// Transition to DURING_MOTION drive mode
rtEnableMode(CLK:=(stMotionStage.nEnableMode = E_StageEnableMode.DURING_MOTION));
// Handle auto-enable timing
CASE stMotionStage.nEnableMode OF
    E_StageEnableMode.ALWAYS:
        stMotionStage.bEnable := TRUE;
    E_StageEnableMode.DURING_MOTION:
        IF rtEnableMode.Q THEN
            stMotionStage.bEnable := FALSE;
        END_IF
        IF bNewMoveReq THEN
            IF stMotionStage.nCommand = E_EpicsMotorCmd.HOME THEN
                stMotionStage.bEnable := stMotionStage.bSafetyReady;
            ELSIF bPosGoal THEN
                IF stMotionStage.bAllForwardEnable THEN
                    stMotionStage.bEnable S= stMotionStage.bSafetyReady;
                ELSIF NOT stMotionStage.bError THEN
                    // Not an error, just a warning
                    stMotionStage.sErrorMessage := 'Cannot move past positive limit.';
                    stMotionStage.bExecute := FALSE;
                END_IF
            ELSIF bNegGoal THEN
                IF stMotionStage.bAllBackwardEnable THEN
                    stMotionStage.bEnable S= stMotionStage.bSafetyReady;
                ELSIF NOT stMotionStage.bError THEN
                    // Not an error, just a warning
                    stMotionStage.sErrorMessage := 'Cannot move past negative limit.';
                    stMotionStage.bExecute := FALSE;
                END_IF
            ELSE
                // Super rare condition where we asked for a move to exactly the same floating point we're already at
                stMotionStage.bEnable S= stMotionStage.bSafetyReady;
            END_IF
            IF stMotionStage.bEnable OR stMotionStage.bError THEN
                bNewMoveReq := FALSE;
            END_IF
        END_IF
END_CASE

// Update all enable booleans
fbSetEnables(stMotionStage:=stMotionStage);

IF stMotionStage.stAxisStatus.bBusy AND NOT bExecute THEN
    // Wait for the previous move to end
    bExecute := FALSE;
ELSIF bMoveCmd THEN
    // Do not start the move until we have power and the safety system says it is OK
    bExecute := stMotionStage.bExecute AND stMotionStage.bAllEnable AND stMotionStage.bEnableDone AND stMotionStage.bSafetyReady;
ELSE
    bExecute := stMotionStage.bExecute;
END_IF

IF bExecute AND NOT stMotionStage.bError THEN
    // Reset local warnings if things are going well
    stMotionStage.sErrorMessage := '';
END_IF

// No moves allowed in error states
IF stMotionStage.bError THEN
    bExecute := FALSE;
END_IF


bExecHome := bExecute AND stMotionStage.nCommand = 10;
bExecMove := bExecute AND NOT bExecHome;

// handles backlash compensention
fbBacklashCompensation(stMotionStage:=stMotionStage,
    bHoming:=bExecHome,
    bMoving:=bExecMove );

// Handle standard commands using ESS's FB
fbDriveVirtual(En:=TRUE,
    bEnable:=stMotionStage.bAllEnable,
    bReset:=stMotionStage.bReset,
    bExecute:=bExecMove,
    nCommand:=INT_TO_UINT(stMotionStage.nCommand),
    nCmdData:=INT_TO_UINT(stMotionStage.nCmdData),
    fVelocity:=stMotionStage.fVelocity,
    fPosition:=stMotionStage.fPosition,
    fAcceleration:=stMotionStage.fAcceleration,
    fDeceleration:=stMotionStage.fDeceleration,
    bLimitFwd:=stMotionStage.bAllForwardEnable,
    bLimitBwd:=stMotionStage.bAllBackwardEnable,
    bHomeSensor:=stMotionStage.bHome,
    fHomePosition:=stMotionStage.fHomePosition,
    bPowerSelf:=stMotionStage.bPowerSelf,
    nMotionAxisID=>stMotionStage.nMotionAxisID,
    Axis:=stMotionStage.Axis);

// Some custom home handling
fbMotionHome(
    stMotionStage:=stMotionStage,
    bExecute:=bExecHome);

// Update status again after the move starts or stops
stMotionStage.Axis.ReadStatus();

// Check for a new error
IF NOT stMotionStage.bError THEN
    stMotionStage.bError := fbDriveVirtual.bError;
    stMotionStage.nErrorId := fbDriveVirtual.nErrorId;
END_IF
IF NOT stMotionStage.bError THEN
    stMotionStage.bError := fbBacklashCompensation.bError;
    stMotionStage.nErrorId := fbBacklashCompensation.nErrorId;
END_IF
IF NOT stMotionStage.bError THEN
    stMotionStage.bError := fbMotionHome.bError;
    stMotionStage.nErrorId := fbMotionHome.nErrorId;
END_IF
IF NOT stMotionStage.bError AND stMotionStage.bExecute AND NOT stMotionStage.bUserEnable THEN
    stMotionStage.bError := TRUE;
    stMotionStage.nErrorId := 1;
    stMotionStage.sCustomErrorMessage := 'Move requested, but user enable is disabled!';
END_IF

// Set the error message if we have one
IF stMotionStage.bError THEN
    // Hook if other code wants to inject a non-NC error
    IF stMotionStage.sCustomErrorMessage <> '' THEN
        stMotionStage.sErrorMessage := stMotionSTage.sCustomErrorMessage;
    ELSE
        stMotionStage.sErrorMessage := F_MotionErrorCodeLookup(nErrorId := stMotionStage.nErrorId);
    END_IF
END_IF

fbLogError(
    stMotionStage:=stMotionStage,
    bEnable:=TRUE);

// When we start, set the busy/done appropriately
rtExec(CLK:=bExecute);
IF rtExec.Q THEN
    stMotionStage.bBusy := TRUE;
    stMotionStage.bDone := FALSE;
END_IF

// Force everything off in case of error
IF stMotionStage.bError THEN
    stMotionStage.bBusy := FALSE;
    stMotionStage.bDone := FALSE;
    stMotionStage.bEnable := FALSE;
END_IF

// Check the limits and cancel execution if appropriate. Without this block we have infinite error spam
bFwdHit := stMotionStage.Axis.Status.PositiveDirection AND NOT stMotionStage.bAllForwardEnable;
bBwdHit := stMotionStage.Axis.Status.NegativeDirection AND NOT stMotionStage.bAllBackwardEnable;
IF (bFwdHit OR bBwdHit) AND NOT fbMotionHome.bBusy THEN
    stMotionStage.bExecute := FALSE;
END_IF

// Check done moving via user stop, fbDriveVirtual and Target Position Monitoring, or from homing.
ftExec(CLK:=stMotionStage.bExecute);
rtTarget(CLK:=(stMotionStage.Axis.Status.InTargetPosition AND fbDriveVirtual.bDone AND bExecMove));
rtHomed(CLK:=fbMotionHome.bDone AND bExecHome);
IF ftExec.Q OR rtTarget.Q OR rtHomed.Q THEN
    IF NOT stMotionStage.bDone THEN
        stMotionStage.bDone := TRUE;
        stMotionStage.bBusy := FALSE;
        IF NOT stMotionStage.Axis.Status.Error THEN
            bExecute := FALSE;
            stMotionStage.bExecute := FALSE;
        END_IF
    END_IF
END_IF

// Handle auto-disable timing
bPrepareDisable S= stMotionStage.nEnableMode = E_StageEnableMode.DURING_MOTION AND ftExec.Q;
// Delay the disable until we reach standstill, else brake issues or other race conditions
IF bPrepareDisable AND stMotionStage.Axis.Status.MotionState = MC_AXISSTATE_STANDSTILL THEN
    bPrepareDisable := FALSE;
    stMotionStage.bEnable := FALSE;
END_IF

// Get a definitive bEnabled reading
CASE stMotionStage.Axis.Status.MotionState OF
    // We are not enabled if there is an issue
    MC_AXISSTATE_UNDEFINED, MC_AXISSTATE_DISABLED, MC_AXISSTATE_ERRORSTOP:
        stMotionStage.bEnableDone := FALSE;
    ELSE
        stMotionStage.bEnableDone := TRUE;
END_CASE

// Handle the brake. TRUE means brake disabled/released
IF stMotionStage.nBrakeMode <> E_StageBrakeMode.NO_BRAKE THEN
    CASE stMotionStage.Axis.Status.MotionState OF
        MC_AXISSTATE_UNDEFINED,
        MC_AXISSTATE_DISABLED,
        MC_AXISSTATE_ERRORSTOP:
            stMotionStage.bBrakeRelease := FALSE;
        MC_AXISSTATE_STANDSTILL:
            IF stMotionStage.nBrakeMode = E_StageBrakeMode.IF_MOVING THEN
                stMotionStage.bBrakeRelease := FALSE;
            ELSE
                stMotionStage.bBrakeRelease := TRUE;
            END_IF
        ELSE
            stMotionStage.bBrakeRelease := TRUE;
    END_CASE
END_IF

// Sync the epics status struct
stMotionStage.stAxisStatus := fbDriveVirtual.stAxisStatus;
stMotionStage.stAxisStatus.bEnabled := stMotionStage.bEnableDone;

// Override homing status, dmov as appropriate
stMotionStage.bHomed := fbMotionHome.bDone AND NOT fbMotionHome.bError;
stMotionStage.stAxisStatus.bHomed := stMotionStage.bHomed;
stMotionStage.stAxisStatus.bExecute := bExecute;
stMotionStage.stAxisStatus.nCommand := 3; // If this is not 3, the IOC stops updating positions during homing

// Fill in auxiliary status info
stMotionStage.fPosDiff := stMotionStage.Axis.NcToPlc.PosDiff;

// Reset everything when bReset is flagged
IF stMotionStage.bReset THEN
    stMotionStage.bEnable := FALSE;
    stMotionStage.bReset := FALSE;
    stMotionStage.bExecute := FALSE;
    stMotionStage.bError := FALSE;
    stMotionStage.nErrorId := 0;
    stMotionStage.sErrorMessage := '';
    stMotionStage.sCustomErrorMessage := '';
    bExecute := FALSE;
END_IF

fbEncoderValue(stMotionStage:=stMotionStage);
fbNCParams(
    stMotionStage:=stMotionStage,
    bEnable:=TRUE,
    tRefreshDelay:=T#1s);

// Save and restore as long as not an absolute encoder
fbSaveRestore(
    stMotionStage:=stMotionStage,
    bEnable:=stMotionStage.nHomingMode <> E_EpicsHomeCmd.NONE);

// Main Motion Status Structure
stMotionStatus.nMotionAxisID    := stMotionStage.Axis.NcToPlc.AxisId;
stMotionStatus.bEnabled         := stMotionStage.bAllEnable;
stMotionStatus.bHomeSensor      := stMotionStage.bHome;
stMotionStatus.bLimitBwd        := stMotionStage.bAllBackwardEnable;
stMotionStatus.bLimitFwd        := stMotionStage.bAllForwardEnable;
stMotionStatus.fActDiff         := stMotionStage.Axis.NcToPlc.PosDiff;
stMotionStatus.fActPosition     := stMotionStage.Axis.NcToPlc.ActPos;
stMotionStatus.fActVelocity     := stMotionStage.Axis.NcToPlc.ActVelo;
stMotionStatus.fOverride        := stMotionStage.Axis.PlcToNc.Override;
stMotionStatus.bBusy            := stMotionStage.bBusy;
stMotionStatus.bHomed           := stMotionStage.bHomed;
stMotionStatus.bWarning         := FALSE; // NOT SUPPORTED BY THIS IMPLEMENTATION
stMotionStatus.bError           := stMotionStage.bError;
stMotionStatus.nErrorId         := stMotionStage.nErrorId;
stMotionStatus.sErrorMessage    := stMotionStage.sErrorMessage;

// Extended Motion Status (Debug, Testing) NOT SUPPORTED BY THIS IMPLEMENTATION
// stExMotionStatus.bMotionAxisError
// stExMotionStatus.nMotionAxisErrorId
// stExMotionStatus.bInterlocksError
// stExMotionStatus.nInterlocksError
// stExMotionStatus.eDriveState
// stExMotionStatus.bAbortDone
// stExMotionStatus.bAborted
// stExMotionStatus.bLimHomeDone
// stExMotionStatus.bDriveWatchDogStatus
// stExMotionStatus.bNewMoveReq
// stExMotionStatus.bEnable
// stExMotionStatus.bIdling

// Main Motion Command Structure
stMotionCmdNow.bHalt := FALSE;
stMotionCmdNow.bHomeCmd := FALSE;
stMotionCmdNow.bMoveCmd := FALSE;
stMotionCmdNow.bReset := FALSE;
stMotionCmdNow.fAcceleration := stMotionStage.fAcceleration;
stMotionCmdNow.fDeceleration := stMotionStage.fDeceleration;
stMotionCmdNow.fHomePosition := stMotionStage.fHomePosition;
//stMotionCmdNow.fJerk := stMotionStage.fJerk; NOT SUPPORTED BY THIS IMPLEMENTATION
stMotionCmdNow.fPosition := stMotionStage.fPosition;
stMotionCmdNow.fVelocity := stMotionStage.fVelocity;
stMotionCmdNow.nCmdData := stMotionStage.nCmdData;
stMotionCmdNow.nCommand := stMotionStage.nCommand;

stMotionCmdPrev := stMotionCmdNow;


METHOD AbsoluteMove
VAR_INPUT
    Position	: LREAL;
    Velocity	: LREAL;
    Acceleration	: LREAL;
    Deceleration	: LREAL;
END_VAR

IF NOT __ISVALIDREF(THIS^.stMotionStageMethods) THEN
    RETURN;
END_IF

THIS^.stMotionStageMethods.fPosition := Position;
THIS^.stMotionStageMethods.fVelocity := Velocity;
THIS^.stMotionStageMethods.fAcceleration := Acceleration;
THIS^.stMotionStageMethods.fDeceleration := Deceleration;
THIS^.stMotionStageMethods.bMoveCmd := TRUE;
END_METHOD


METHOD AbsoluteMoveWithBacklashCompensation
VAR_INPUT
    Position	: LREAL;
    Velocity	: LREAL;
    Acceleration	: LREAL;
    Deceleration	: LREAL;
END_VAR

IF NOT __ISVALIDREF(THIS^.stMotionStageMethods) THEN
    RETURN;
END_IF

THIS^.stMotionStageMethods.fPosition := Position;
THIS^.stMotionStageMethods.fVelocity := Velocity;
THIS^.stMotionStageMethods.fAcceleration := Acceleration;
THIS^.stMotionStageMethods.fDeceleration := Deceleration;
THIS^.stMotionStageMethods.bMoveCmd := TRUE;
END_METHOD


PROPERTY BrakeMode : LCLS_OOPMotion.E_StageBrakeMode
GET

CASE THIS^.stMotionStageMethods.nBrakeMode OF
    E_StageBrakeMode.NO_BRAKE:
        BrakeMode := LCLS_OOPMotion.E_StageBrakeMode.NO_BRAKE;
    E_StageBrakeMode.IF_MOVING:
        BrakeMode := LCLS_OOPMotion.E_StageBrakeMode.IF_MOVING;
    E_StageBrakeMode.IF_ENABLED:
        BrakeMode := LCLS_OOPMotion.E_StageBrakeMode.IF_ENABLED;
END_CASE
END_GET
SET

CASE BrakeMode OF
    LCLS_OOPMotion.E_StageBrakeMode.NO_BRAKE:
        THIS^.stMotionStageMethods.nBrakeMode := E_StageBrakeMode.NO_BRAKE;
    LCLS_OOPMotion.E_StageBrakeMode.IF_MOVING:
        THIS^.stMotionStageMethods.nBrakeMode := E_StageBrakeMode.IF_MOVING;
    LCLS_OOPMotion.E_StageBrakeMode.IF_ENABLED:
        THIS^.stMotionStageMethods.nBrakeMode := E_StageBrakeMode.IF_ENABLED;
END_CASE
END_SET
END_PROPERTY


PROPERTY EnableMode : LCLS_OOPMotion.E_StageEnableMode
GET

CASE THIS^.stMotionStageMethods.nEnableMode OF
    E_StageEnableMode.ALWAYS:
        EnableMode := LCLS_OOPMotion.E_StageEnableMode.ALWAYS;
    E_StageEnableMode.DURING_MOTION:
        EnableMode := LCLS_OOPMotion.E_StageEnableMode.DURING_MOTION;
    E_StageEnableMode.NEVER:
        EnableMode := LCLS_OOPMotion.E_StageEnableMode.NEVER;
END_CASE
END_GET
SET

CASE EnableMode OF
    LCLS_OOPMotion.E_StageEnableMode.ALWAYS:
        THIS^.stMotionStageMethods.nEnableMode := E_StageEnableMode.ALWAYS;
    LCLS_OOPMotion.E_StageEnableMode.DURING_MOTION:
        THIS^.stMotionStageMethods.nEnableMode := E_StageEnableMode.DURING_MOTION;
    LCLS_OOPMotion.E_StageEnableMode.NEVER:
        THIS^.stMotionStageMethods.nEnableMode := E_StageEnableMode.NEVER;
END_CASE
END_SET
END_PROPERTY


PROPERTY ExMotionStatus : REFERENCE TO LCLS_OOPMotion.ST_ExtendedMotionStatus
GET

ExMotionStatus REF= THIS^.stExMotionStatus;
END_GET
END_PROPERTY


METHOD Halt

IF NOT __ISVALIDREF(THIS^.stMotionStageMethods) THEN
    RETURN;
END_IF

THIS^.stMotionStageMethods.bExecute := FALSE;
END_METHOD


METHOD Home
VAR_INPUT
    HomePosition	: LREAL;
    HomeMode	: INT;
END_VAR

IF NOT __ISVALIDREF(THIS^.stMotionStageMethods) THEN
    RETURN;
END_IF

THIS^.stMotionStageMethods.fHomePosition := HomePosition;

CASE HomeMode OF
    E_EpicsHomeCmd.ABSOLUTE_SET:
        THIS^.stMotionStageMethods.nHomingMode := E_EpicsHomeCmd.ABSOLUTE_SET;
    E_EpicsHomeCmd.AutoMethod:
        THIS^.stMotionStageMethods.nHomingMode := E_EpicsHomeCmd.AutoMethod;
    E_EpicsHomeCmd.CURRENT_POSITION_METHOD:
        THIS^.stMotionStageMethods.nHomingMode := E_EpicsHomeCmd.CURRENT_POSITION_METHOD;
    E_EpicsHomeCmd.HIGH_LIMIT:
        THIS^.stMotionStageMethods.nHomingMode := E_EpicsHomeCmd.HIGH_LIMIT;
    E_EpicsHomeCmd.HOME_VIA_HIGH:
        THIS^.stMotionStageMethods.nHomingMode := E_EpicsHomeCmd.HOME_VIA_HIGH;
    E_EpicsHomeCmd.HOME_VIA_LOW:
        THIS^.stMotionStageMethods.nHomingMode := E_EpicsHomeCmd.HOME_VIA_LOW;
    E_EpicsHomeCmd.LOW_LIMIT:
        THIS^.stMotionStageMethods.nHomingMode := E_EpicsHomeCmd.LOW_LIMIT;
    E_EpicsHomeCmd.NONE:
        THIS^.stMotionStageMethods.nHomingMode := E_EpicsHomeCmd.NONE;
END_CASE

THIS^.stMotionStageMethods.bHomeCmd := TRUE;
END_METHOD


PROPERTY MotionCmd : REFERENCE TO LCLS_OOPMotion.ST_MotionCommand
GET

MotionCmd REF= THIS^.stMotionCmdNow;
END_GET
END_PROPERTY


PROPERTY MotionStatus : REFERENCE TO LCLS_OOPMotion.ST_MotionStatus
GET

MotionStatus REF= THIS^.stMotionStatus;
END_GET
END_PROPERTY


METHOD Reset

IF NOT __ISVALIDREF(THIS^.stMotionStageMethods) THEN
    RETURN;
END_IF

THIS^.stMotionStageMethods.bReset := TRUE;
END_METHOD


PROPERTY SaveAxisParams : BOOL
SET

// NOT SUPPORTED BY THIS IMPLEMENTATION
END_SET
END_PROPERTY


METHOD StateMove
VAR_INPUT
    Execute	: BOOL;
END_VAR

IF NOT __ISVALIDREF(stMotionStageMethods) THEN
    RETURN;
END_IF
END_METHOD

END_FUNCTION_BLOCK

// ---- POUs/Motion/FB_MotionHoming.TcPOU
FUNCTION_BLOCK FB_MotionHoming
VAR_IN_OUT
    stMotionStage: ST_MotionStage;
END_VAR
VAR_INPUT
    bExecute: BOOL;
END_VAR
VAR_OUTPUT
    bBusy: BOOL;
    bDone: BOOL;
    bError: BOOL;
    nErrorID: UDINT;
END_VAR
VAR
    fbSetPos: MC_SetPosition;
    fbJog: MC_Jog;
    rtExec: R_TRIG;
    ftExec: F_TRIG;
    nHomeStateMachine: INT := IDLE;
    nStateAfterStop: INT;
    nMoves: INT;
    bFirstDirection: BOOL;
    bAtHome: BOOL;
    bMove: BOOL;
    nErrCount: INT;
    bInterrupted: BOOL;
END_VAR
VAR CONSTANT
    IDLE: INT := 0;
    NEXT_MOVE: INT := 1;
    CHECK_FWD: INT := 2;
    CHECK_BWD: INT := 3;
    FINAL_MOVE: INT := 4;
    FINAL_SETPOS: INT := 5;
    ERROR: INT := 6;
    WAIT_STOP: INT := 7;

    (*
        This is a simpler way of disabling the soft limits that ends up being really obvious if something has gone wrong.
        If you turn the limits off/on, not only do you need to keep track of if you had soft limits set,
        but you need to always restore this properly or risk some issue.
        Instead, I set position to a ridiculous value that can always move forward or backward.
        If this gets stuck for any reason it's very clear that something has gone wrong,
        rather than a silent failure of the soft limit marks.
    *)
    FWD_START: LREAL := -99999999;
    BWD_START: LREAL :=  99999999;
END_VAR


fbSetPos.Options.ClearPositionLag := TRUE;
rtExec(CLK:=bExecute);
ftExec(CLK:=bExecute);

bError R= NOT bExecute;
IF NOT bError THEN
    nErrorID := 0;
END_IF

CASE stMotionStage.nHomingMode OF
    E_EpicsHomeCmd.LOW_LIMIT:
        bFirstDirection := FALSE;
        bAtHome := NOT stMotionStage.bLimitBackwardEnable;
        bMove := TRUE;
    E_EpicsHomeCmd.HIGH_LIMIT:
        bFirstDirection := TRUE;
        bAtHome := NOT stMotionStage.bLimitForwardEnable;
        bMove := TRUE;
    E_EpicsHomeCmd.HOME_VIA_LOW:
        bFirstDirection := FALSE;
        bAtHome := stMotionStage.bHome;
        bMove := TRUE;
    E_EpicsHomeCmd.HOME_VIA_HIGH:
        bFirstDirection := TRUE;
        bAtHome := stMotionStage.bHome;
        bMove := TRUE;
    E_EpicsHomeCmd.ABSOLUTE_SET:
        fbSetPos(
            Axis:=stMotionStage.Axis,
            Execute:=bExecute,
            Position:=stMotionStage.fHomePosition);
        bBusy := rtExec.Q;
        bDone := NOT rtExec.Q;
        bMove := FALSE;
    E_EpicsHomeCmd.NONE:
        bMove := FALSE;
        bBusy := rtExec.Q;
        bDone := NOT rtExec.Q;
    ELSE
        bMove := FALSE;
END_CASE

IF bMove THEN
    IF bBusy AND ftExec.Q THEN
        nHomeStateMachine := ERROR;
        bInterrupted := TRUE;
    END_IF
    CASE nHomeStateMachine OF
        // Wait for a rising edge
        IDLE:
            bBusy := FALSE;
            nErrCount := 0;
            fbSetPos(
                Axis:=stMotionStage.Axis,
                Execute:=FALSE);
            fbJog(
                Axis:=stMotionStage.Axis,
                JogForward:=FALSE,
                JogBackwards:=FALSE);
            IF rtExec.Q THEN
                nHomeStateMachine := NEXT_MOVE;
                nMoves := 0;
                bDone := FALSE;
                bBusy := TRUE;
                bError := FALSE;
                nErrorID := 0;
                bInterrupted := FALSE;
            END_IF
        // Figure out whether to move forward, move backward, or give up
        NEXT_MOVE:
            fbSetPos(
                Axis:=stMotionStage.Axis,
                Execute:=FALSE);
            fbJog(
                Axis:=stMotionStage.Axis,
                JogForward:=FALSE,
                JogBackwards:=FALSE);
            CASE nMoves OF
                0:
                    IF bFirstDirection THEN
                        nStateAfterStop := CHECK_FWD;
                    ELSE
                        nStateAfterStop := CHECK_BWD;
                    END_IF
                1:
                    IF NOT bFirstDirection THEN
                        nStateAfterStop := CHECK_FWD;
                    ELSE
                        nStateAfterStop := CHECK_BWD;
                    END_IF
                ELSE
                    nStateAfterStop := ERROR;
            END_CASE
            nMoves := nMoves + 1;
            IF bAtHome THEN
                nStateAfterStop := FINAL_MOVE;
            END_IF
            nHomeStateMachine := WAIT_STOP;
        // Move forward until we find the home signal or reach end of travel
        CHECK_FWD:
            fbSetPos(
                Axis:=stMotionStage.Axis,
                Execute:=TRUE,
                Position:=FWD_START);
            fbJog(
                Axis:=stMotionStage.Axis,
                JogForward:=stMotionStage.bLimitForwardEnable AND NOT bATHome,
                JogBackwards:=FALSE,
                Mode:=E_JogMode.MC_JOGMODE_CONTINOUS,
                Velocity:=stMotionStage.stAxisParameters.fRefVeloSearch);
            IF NOT fbJog.JogForward THEN
                nHomeStateMachine := NEXT_MOVE;
            ELSIF fbJog.Error THEN
                fbJog(
                    Axis:=stMotionStage.Axis,
                    JogForward:=FALSE,
                    JogBackwards:=FALSE);
                nErrCount := nErrCount + 1;
                IF nErrCount >= 3 THEN
                    nHomeStateMachine := ERROR;
                END_IF
            END_IF
        // Move backward until we find the home signal or reach end of travel
        CHECK_BWD:
            fbSetPos(
                Axis:=stMotionStage.Axis,
                Execute:=TRUE,
                Position:=BWD_START);
            fbJog(
                Axis:=stMotionStage.Axis,
                JogForward:=FALSE,
                JogBackwards:=stMotionStage.bLimitBackwardEnable AND NOT bATHome,
                Mode:=E_JogMode.MC_JOGMODE_CONTINOUS,
                Velocity:=stMotionStage.stAxisParameters.fRefVeloSearch);
            IF NOT fbJog.JogBackwards THEN
                nHomeStateMachine := NEXT_MOVE;
            ELSIF fbJog.Error THEN
                fbJog(
                    Axis:=stMotionStage.Axis,
                    JogForward:=FALSE,
                    JogBackwards:=FALSE);
                nErrCount := nErrCount + 1;
                IF nErrCount >= 3 THEN
                    nHomeStateMachine := ERROR;
                END_IF
            END_IF
        // Set position to get within soft lims, move slowly off signal
        FINAL_MOVE:
            fbSetPos(
                Axis:=stMotionStage.Axis,
                Execute:=TRUE,
                Position:=stMotionStage.fHomePosition);
            IF bAtHome THEN
                fbJog(
                    Axis:=stMotionStage.Axis,
                    JogForward:=NOT bFirstDirection,
                    JogBackwards:=bFirstDirection,
                    Mode:=E_JogMode.MC_JOGMODE_CONTINOUS,
                    Velocity:=stMotionStage.stAxisParameters.fRefVeloSync);
            ELSIF fbJog.Error THEN
                fbJog(
                    Axis:=stMotionStage.Axis,
                    JogForward:=FALSE,
                    JogBackwards:=FALSE);
                nErrCount := nErrCount + 1;
                IF nErrCount >= 3 THEN
                    nHomeStateMachine := ERROR;
                END_IF
            ELSE
                fbJog(
                    Axis:=stMotionStage.Axis,
                    JogForward:=FALSE,
                    JogBackwards:=FALSE);
                fbSetPos(
                    Axis:=stMotionStage.Axis,
                    Execute:=FALSE);
                nHomeStateMachine := WAIT_STOP;
                nStateAfterStop := FINAL_SETPOS;
            END_IF
        FINAL_SETPOS:
            fbSetPos(
                Axis:=stMotionStage.Axis,
                Execute:=TRUE,
                Position:=stMotionStage.fHomePosition);
            nHomeStateMachine := IDLE;
            bBusy := FALSE;
            bDone := TRUE; // need this
        ERROR:
            bError := TRUE;
            nErrorID := fbJog.ErrorID;
            nHomeStateMachine := FINAL_SETPOS;
            fbSetPos(
                Axis:=stMotionStage.Axis,
                Execute:=FALSE);
            IF bInterrupted THEN
                stMotionStage.sCustomErrorMessage := 'Homing interrupted';
            ELSE
                stMotionStage.sCustomErrorMessage := 'Homing failure';
            END_IF
        WAIT_STOP:
            IF stMotionStage.Axis.Status.NotMoving THEN
                nHomeStateMachine := nStateAfterStop;
            END_IF
    END_CASE
END_IF

END_FUNCTION_BLOCK

// ---- POUs/Motion/FB_EncSaveRestore.TcPOU
FUNCTION_BLOCK FB_EncSaveRestore
VAR_IN_OUT
    stMotionStage: ST_MotionStage;
END_VAR
VAR_INPUT
    bEnable: BOOL;
END_VAR
VAR_OUTPUT
END_VAR
VAR
    fbSetPos: MC_SetPosition;
    timer: TON;
    bInit: BOOL;
    bLoad: BOOL;
    nLatchError: UDINT;
    bEncError: BOOL;
    tRetryDelay: TIME := T#1s;
    nMaxRetries: UINT := 10;
    nCurrTries: UINT := 0;
    bWaitRetry: BOOL;
    tonRetry: TON;
END_VAR
VAR PERSISTENT
    bSaved: BOOL;
    fPosition: LREAL;
END_VAR

IF bEnable THEN
    // Trigger a load if anything was saved at all
    IF NOT bInit THEN
        bInit := TRUE;
        bLoad S= bSaved;
        fbSetPos.Options.ClearPositionLag := TRUE;
    END_IF

    // Set our position if bLoad is true
    fbSetPos(
        Axis:=stMotionStage.Axis,
        Execute:=bLoad,
        Position:=fPosition);

    // Only load once, at startup
    bLoad R= fbSetPos.Done OR fbSetPos.Error;

    IF fbSetPos.Error THEN
        // Keep the error latched, it can disappear if Execute is set to FALSE
        nLatchError := fbSetPos.ErrorID;
        nCurrTries := nCurrTries + 1;
        IF nCurrTries >= nMaxRetries THEN
            // Alert the user that something has gone wrong
            stMotionStage.bError := TRUE;
            stMotionStage.nErrorId := nLatchError;
            stMotionStage.sCustomErrorMessage := 'Error loading previously saved position.';
        ELSE
            // Reset the FB for the next retry
            fbSetPos(
                Axis:=stMotionStage.Axis,
                Execute:=FALSE,
                Position:=fPosition);
            // Try again
            bWaitRetry := TRUE;
        END_IF
    END_IF

    tonRetry(
        IN := bWaitRetry,
        PT := tRetryDelay);

    bLoad S= tonRetry.Q;
    bWaitRetry R= tonRetry.Q;

    // Check ST_MotionStage for an encoder error (range 0x44nn)
    bEncError := stMotionStage.bError AND stMotionStage.nErrorId >= 16#4400 AND stMotionStage.nErrorId <= 16#44FF;

    // Do not save if we're currently loading or if there is an encoder error
    IF NOT bLoad AND NOT bEncError AND NOT bWaitRetry THEN
        fPosition := stMotionStage.stAxisStatus.fActPosition;
        // This persistent variable lets us check if anything was saved
        // It will be TRUE at startup if we have saved values
        bSaved := TRUE;
    END_IF
END_IF

END_FUNCTION_BLOCK

// ---- POUs/Motion/FB_LogMotionError.TcPOU
FUNCTION_BLOCK FB_LogMotionError
(*
    If the motion struct has an error, log it.

    The log condition is:
    - When bError goes TRUE (catch transition from no error to error)
    - When the error message changes while bError is TRUE (catch transition from error a to error b)

    Includes the motor name and the NC error id in the json blob
*)
VAR_IN_OUT
    stMotionStage: ST_MotionStage;
END_VAR
VAR_INPUT
    bEnable: BOOL;
END_VAR
VAR
    fbLogMessage: FB_LogMessage;
    rtNewError: R_TRIG;
    bChangedError: BOOL;
    sPrevErr: STRING;
    fbJson: FB_JsonSaxWriter;
END_VAR


rtNewError(CLK:=stMotionStage.bError);
bChangedError := stMotionStage.sErrorMessage <> '' AND stMotionStage.sErrorMessage <> sPrevErr;
sPrevErr := stMotionStage.sErrorMessage;

IF bEnable AND (rtNewError.Q OR bChangedError) THEN
    fbJson.StartObject();
    fbJson.AddKey('schema');
    fbJson.AddString('ST_MotionStage.bError');
    fbJson.AddKey('dut_name');
    fbJson.AddString(stMotionStage.sName);
    fbJson.AddKey('axis_name');
    fbJson.AddString(stMotionStage.stAxisParameters.sAxisName);
    fbJson.AddKey('axis_id');
    fbJson.AddUdint(stMotionStage.stAxisParameters.AxisId);
    fbJson.AddKey('err_id');
    fbJson.AddUdint(stMotionStage.nErrorId);
    fbJson.AddKey('position');
    fbJson.AddLreal(stMotionStage.stAxisStatus.fActPosition);
    fbJson.AddKey('position_lag');
    fbJson.AddLreal(stMotionStage.stAxisStatus.fActDiff);
    fbJson.EndObject();
    fbLogMessage.sJson := fbJson.GetDocument();
    fbLogMessage(
        sMsg := stMotionStage.sErrorMessage,
        eSevr := TcEventSeverity.Error,
        eSubsystem := E_Subsystem.MOTION,
    );
    fbJson.ResetDocument();
END_IF

END_FUNCTION_BLOCK

// ---- POUs/Motion/FB_MotionBacklashCompensation.TcPOU
FUNCTION_BLOCK FB_MotionBacklashCompensation
(*
    Handle positive/negative backlash compensation
    User needs to set the direction of backlash from the sign of the compensation value
    Backlash compensation is disabled during referencing (homing).
    When direction is positive/negative, further movement in the negative/positive direction not compensated
    further movement in the negative/positive direction will be compensated
*)
VAR_IN_OUT
    stMotionStage: ST_MotionStage;
END_VAR
VAR_INPUT
    bHoming: BOOL;
    bMoving: BOOL;
END_VAR
VAR_OUTPUT
    bError: BOOL;
    nErrorID: UDINT;
END_VAR
VAR
    fbBacklashCompensation: MC_BacklashCompensation;
    fPrevCompensation : LREAL := 0.0;
    bBacklashCompEnable: BOOL;
END_VAR

(*Note: Configure within the axis parameters set "position correction" to true *)
(*Directional change for compensation
  default: positive backlash):
  TRUE -> Negative backlash compensation *)
(* Reset Compensation to register a new value change*)
bBacklashCompEnable R= bHoming OR (stMotionStage.fBacklash<>fPrevCompensation);
bBacklashCompEnable S= bMoving;

fbBacklashCompensation(Axis:=stMotionStage.Axis,
    Enable:= ( stMotionStage.bUserBacklashEn AND bBacklashCompEnable),
    Backlash:=stMotionStage.fBacklash,
    CompensationInPositiveDirection:=(stMotionStage.fBacklash<0.0),
    Ramp:=(stMotionStage.fVelocity / 10.0),
    DisableMode:=DisableModeHold,
    Enabled=> stMotionStage.bBacklashStatus,
    Error=>bError,
    ErrorID=>nErrorID,
    CurrentBacklash=>stMotionStage.fCurrentBacklash);

fPrevCompensation:=stMotionStage.fBacklash;

END_FUNCTION_BLOCK

// ---- POUs/Motion/Utils/FB_SetEnables.TcPOU
FUNCTION_BLOCK FB_SetEnables
// Update the all enable booleans based on the booleans that make them up
VAR_IN_OUT
    stMotionStage: ST_MotionStage;
END_VAR

stMotionStage.bAllForwardEnable := stMotionStage.bLimitForwardEnable AND (stMotionStage.bGantryForwardEnable OR NOT stMotionStage.bGantryAxis) AND stMotionStage.stEPSForwardEnable.bEPS_OK;
stMotionStage.bAllBackwardEnable := stMotionStage.bLimitBackwardEnable AND (stMotionStage.bGantryBackwardEnable OR NOT stMotionStage.bGantryAxis) AND stMotionStage.stEPSBackwardEnable.bEPS_OK;

stMotionStage.bAllEnable := stMotionStage.bEnable AND stMotionStage.bHardwareEnable AND stMotionStage.stEPSPowerEnable.bEPS_OK;
stMotionStage.bAllEnable R= NOT stMotionStage.bUserEnable;

END_FUNCTION_BLOCK

// ---- POUs/Motion/FB_EncoderValue.TcPOU
FUNCTION_BLOCK FB_EncoderValue
(*
    Process the encoder value for ST_MotionStage

    A few different problems this is trying to solve:
        1. Different encoders show as different types in the IO,
           but we want a consistent type for checks and for PVs
        2. Some inverted encoders display as very high numbers
           as they count down from max int instead of up from 0
        3. Some encoders have raw signed values, others unsigned.

    To this end, we figure out which encoder is linked and process
    the value appropriately.
*)
VAR_IN_OUT
    stMotionStage: ST_MotionStage;
END_VAR

IF stMotionStage.nRawEncoderULINT <> 0 THEN
    IF stMotionStage.nRawEncoderULINT < 4294967296 THEN
        stMotionStage.nEncoderCount := ULINT_TO_UDINT(stMotionStage.nRawEncoderULINT);
    ELSE
        stMotionStage.nEncoderCount := ULINT_TO_UDINT(18446744073709551615 - stMotionStage.nRawEncoderULINT);
    END_IF
ELSIF stMotionStage.nRawEncoderUINT <> 0 THEN
    stMotionStage.nEncoderCount := UINT_TO_UDINT(stMotionStage.nRawEncoderUINT);
ELSIF stMotionStage.nRawEncoderINT <> 0 THEN
    stMotionStage.nEncoderCount := INT_TO_UDINT(stMotionStage.nRawEncoderINT);
ELSIF stMotionStage.nRawEncoderDINT <> 0 THEN
    stMotionStage.nEncoderCount := DINT_TO_UDINT(stMotionStage.nRawEncoderDINT);
ELSE
    stMotionStage.nEncoderCount := 0;
END_IF

END_FUNCTION_BLOCK

// ---- POUs/Motion/FB_MotionStageNCParams.TcPOU
FUNCTION_BLOCK FB_MotionStageNCParams
(*
    Read and refresh axis parameters struct on ST_MotionStage
*)
VAR_IN_OUT
    stMotionStage: ST_MotionStage;
END_VAR
VAR_INPUT
    bEnable: BOOL;
    tRefreshDelay: TIME;
END_VAR
VAR_OUTPUT
    bError: BOOL;
END_VAR
VAR
    mcReadParams: MC_ReadParameterSet;
    timer: TON;
    bExecute: BOOL := TRUE;
    nLatchErrId: UDINT;
END_VAR

timer(
    IN:=bEnable AND NOT bExecute,
    PT:=tRefreshDelay);
bExecute S= timer.Q;
mcReadParams(
    Parameter:=stMotionStage.stAxisParameters,
    Axis:=stMotionStage.Axis,
    Execute:=bEnable AND bExecute,
    Error=>bError);

// Copy axis parameters that we want to expose to the EPICS layer.
stMotionStage.stAxisParametersExposed.bCtrlEnablePosDiffControl     := stMotionStage.stAxisParameters.bCtrlEnablePosDiffControl;
stMotionStage.stAxisParametersExposed.bEncEnableSoftEndMaxControl   := stMotionStage.stAxisParameters.bEncEnableSoftEndMaxControl;
stMotionStage.stAxisParametersExposed.bEncEnableSoftEndMinControl   := stMotionStage.stAxisParameters.bEncEnableSoftEndMinControl;
stMotionStage.stAxisParametersExposed.fAccelerationMax              := stMotionStage.stAxisParameters.fAccelerationMax;
stMotionStage.stAxisParametersExposed.fCtrlPosDiffMax               := stMotionStage.stAxisParameters.fCtrlPosDiffMax;
stMotionStage.stAxisParametersExposed.fCtrlPosDiffMaxTime           := stMotionStage.stAxisParameters.fCtrlPosDiffMaxTime;
stMotionStage.stAxisParametersExposed.fDecelerationMax              := stMotionStage.stAxisParameters.fDecelerationMax;
stMotionStage.stAxisParametersExposed.fEncSoftEndMax                := stMotionStage.stAxisParameters.fEncSoftEndMax;
stMotionStage.stAxisParametersExposed.fEncSoftEndMin                := stMotionStage.stAxisParameters.fEncSoftEndMin;
stMotionStage.stAxisParametersExposed.fVeloMaximum                  := stMotionStage.stAxisParameters.fVeloMaximum;
stMotionStage.stAxisParametersExposed.fEncOffset               		:= stMotionStage.stAxisParameters.fEncOffset;
stMotionStage.stAxisParametersExposed.fEncScaleFactorInternal       := stMotionStage.stAxisParameters.fEncScaleFactorInternal;

IF mcReadParams.ErrorID <> 0 THEN
    nLatchErrId := 0;
END_IF
bExecute R= mcReadParams.Done OR mcReadParams.Error;
stMotionStage.bAxisParamsInit S= mcReadParams.Done;

END_FUNCTION_BLOCK

// ---- POUs/Motion/Utils/F_MotionErrorCodeLookup.TcPOU
FUNCTION F_MotionErrorCodeLookup : STRING
VAR_INPUT
    nErrorId: UDINT;
END_VAR
VAR
    msg: STRING;
END_VAR

CASE nErrorId OF
    // General NC Errors
    16#4000: msg:='Internal error';
    16#4001: msg:='Memory error';
    16#4002: msg:='Nc retain data error (persistent data)';
    16#4003: msg:='Parameter for Monitoring the NC Setpoint Issuing is Invalid';
    16#4004: msg:='External Error';
    16#4010: msg:='Channel identifier not allowed';
    16#4011: msg:='Group identifier not allowed';
    16#4012: msg:='Axis identifier not allowed';
    16#4013: msg:='Encoder identifier not allowed';
    16#4014: msg:='Controller identifier not allowed';
    16#4015: msg:='Drive identifier not allowed';
    16#4016: msg:='Table identifier not allowed';
    16#4020: msg:='No process image: No PLC-axis interface';
    16#4021: msg:='No process image: No axis-PLC interface';
    16#4022: msg:='No process image: No encoder-I/O interface';
    16#4023: msg:='No process image: No I/O-encoder interface';
    16#4024: msg:='No process image: No drive-I/O interface';
    16#4025: msg:='No process image: No I/O-drive interface';
    16#4030: msg:='Coupling type not allowed';
    16#4031: msg:='Axis type not allowed';
    16#4032: msg:='Unknown Channel Type';
    16#4040: msg:='Axis is incompatible';
    16#4050: msg:='Channel not ready for operation';
    16#4051: msg:='Group not ready for operation';
    16#4052: msg:='Axis not ready for operation';
    16#4060: msg:='Channel exists';
    16#4061: msg:='Group exists';
    16#4062: msg:='Axis exists';
    16#4063: msg:='Table exists';
    16#4070: msg:='Axis index not allowed';
    16#4071: msg:='Axis index not allowed (group)';

    // Channel Errors
    16#4101: msg:='Group index not allowed';
    16#4102: msg:='Null pointer to group';
    16#4103: msg:='No process image for PLC exchange';
    16#4104: msg:='M-function index not allowed';
    16#4105: msg:='No memory';
    16#4106: msg:='Not ready';
    16#4107: msg:='Function/command not supported';
    16#4108: msg:='Invalid parameter while starting';
    16#4109: msg:='Channel function/command not executable';
    16#410A: msg:='ItpGoAhead not executable';
    16#4110: msg:='Error opening a file';
    16#4111: msg:='Syntax error during loading';
    16#4112: msg:='Syntax error during interpretation';
    16#4113: msg:='Missing subroutine';
    16#4114: msg:='Loading buffer of interpreter is too small';
    16#4117: msg:='Subroutine incomplete';
    16#4118: msg:='Error while loading the NC program';
    16#4119: msg:='Program name too long';
    16#4120: msg:='Divide by zero';
    16#4121: msg:='Invalid circle parameterization';
    16#4122: msg:='Invalid FPU-Operation';
    16#4130: msg:='Stack overflow: subroutines';
    16#4131: msg:='Stack underflow: subroutines';
    16#4132: msg:='Stack overflow: arithmetic unit';
    16#4133: msg:='Stack underflow: arithmetic unit';
    16#4140: msg:='Register index not allowed';
    16#4141: msg:='Unacceptable G-function index';
    16#4142: msg:='Unacceptable M-function index';
    16#4143: msg:='Unacceptable extended address';
    16#4144: msg:='Unacceptable index to internal H-function';
    16#4145: msg:='Machine data value unacceptable';
    16#4150: msg:='Cannot change tool params here';
    16#4151: msg:='Cannot calculate tool compensation';
    16#4152: msg:='Tool compensation: plane cannot be changed here';
    16#4153: msg:='Tool compensation: D-Word missing or invalid';
    16#4154: msg:='Tool compensation: tool radius invalid';
    16#4155: msg:='Tool compensation: tool radius cannot be changed here';
    16#4156: msg:='Tool compensation: Collision Detection Table full';
    16#4157: msg:='Tool compensation: internal error turning on contour collision detection';
    16#4158: msg:='Tool compensation: internal error in contour collision detection';
    16#4159: msg:='Tool compensation: unexpected combination of geometry types';
    16#415A: msg:='Tool compensation: programmed inner circle smaller than cutter radius';
    16#415B: msg:='Tool compensation: bottle neck detection recognized contour violation';
    16#415C: msg:='Table for corrected entries is full';
    16#415D: msg:='Input table for tangential following is full';
    16#415E: msg:='Executing table for tangential following is full';
    16#415F: msg:='Geometric entry for tangential following cannot be calculated';
    16#4162: msg:='Active interpolation rules cannot be detected';
    16#4170: msg:='Error while loading: Invalid parameter';
    16#4171: msg:='Invalid contour start position';
    16#4172: msg:='Retrace: Invalid internal entry index';
    16#4173: msg:='Invalid G Code';
    16#4174: msg:='Error while Opening the G Code File';

    // Group Errors
    16#4200: msg:='Group ID not allowed';
    16#4201: msg:='Group type not allowed';
    16#4202: msg:='Master axis index not allowed';
    16#4203: msg:='Slave axis index not allowed';
    16#4204: msg:='Internal Error';
    16#4205: msg:='Invalid cycle time for SAF';
    16#4206: msg:='GROUPERR_RANGE_MAXELEMENTSINAXIS';
    16#4207: msg:='Invalid cycle time for SVB';
    16#4208: msg:='Single step mode not allowed';
    16#4209: msg:='Group deactivation not allowed';
    16#420A: msg:='SAF state not allowed';
    16#420B: msg:='Channel address invalid';
    16#420C: msg:='Axis address (master axis) invalid';
    16#420D: msg:='Master axis address invalid';
    16#420E: msg:='Slave axis address invalid';
    16#420F: msg:='Slave set value generator address invalid';
    16#4210: msg:='Encoder address invalid';
    16#4211: msg:='Controller address invalid';
    16#4212: msg:='Drive address invalid';
    16#4213: msg:='Address Master Setpoint Generator invalid';
    16#4214: msg:='Axis interface NC to PLC address invalid';
    16#4215: msg:='Slave axis address invalid';
    16#4216: msg:='Table address unknown';
    16#4217: msg:='NcControl address invalid';
    16#4218: msg:='Axis blocked for commands while persistent NC data queued';
    16#4219: msg:='Scaling mode MASTER-AUTOOFFSET invalid';
    16#421A: msg:='Master axis start position does not permit synchronization';
    16#421B: msg:='Slave coupling factor of 0.0 is not allowed';
    16#421C: msg:='Insertion of master axis into group not allowed';
    16#421D: msg:='Deletion of master axis from group not allowed';
    16#421E: msg:='Function/feature not supported from setpoint generator';
    16#421F: msg:='Group initialization';
    16#4220: msg:='Group not ready for new task';
    16#4221: msg:='Requested set velocity is not allowed';
    16#4222: msg:='Requested set position is not allowed';
    16#4223: msg:='No enable for controller and/or feed';
    16#4224: msg:='Movement smaller than one encoder increment';
    16#4225: msg:='Drive not ready during axis start';
    16#4226: msg:='Invalid parameters of emergency stop';
    16#4227: msg:='Setpoint generator is inactive';
    16#4228: msg:='Requested traverse distance is not allowed';
    16#4229: msg:='Requested target position not allowed (slave axis)';
    16#422A: msg:='No enable for controller and/or feed (slave axis)';
    16#422B: msg:='Activation position out of range';
    16#422C: msg:='Start or activation data of external setpoint generation not valid';
    16#422D: msg:='Velocity is not constant';
    16#422E: msg:='Jerk less than or equal to 0.0 is not allowed';
    16#422F: msg:='Acceleration less than or equal to 0.0 is not allowed';
    16#4230: msg:='Deceleration less than or equal to 0.0 is not allowed';
    16#4231: msg:='Set velocity less than or equal to 0.0 is not allowed';
    16#4232: msg:='Loss of precision when trying positioning';
    16#4233: msg:='Cycle time less than or equal to 0.0 is not allowed';
    16#4234: msg:='PTP data type intasdouble range exceeded';
    16#4235: msg:='PTP LHL velocity profile cannot be generated';
    16#4236: msg:='PTP HML velocity profile cannot be generated';
    16#4237: msg:='Start data address is invalid';
    16#4238: msg:='Velocity override not allowed';
    16#4239: msg:='Start type not allowed';
    16#423A: msg:='Velocity overflow';
    16#423B: msg:='Start parameter for axis structure invalid';
    16#423C: msg:='Override generator initialization parameter invalid';
    16#423D: msg:='Slave axis has no set value generator';
    16#423E: msg:='Table is empty';
    16#423F: msg:='Table is full';
    16#4240: msg:='No memory available';
    16#4241: msg:='Table already contains an entry';
    16#4242: msg:='Stop is already active';
    16#4243: msg:='Compensation has not been carried out over full section';
    16#4244: msg:='Internal parameters for compensation are invalid';
    16#4245: msg:='Compensation active';
    16#4246: msg:='Compensation not active';
    16#4247: msg:='Compensation type invalid';
    16#4248: msg:='Axis address for compensation invalid';
    16#4249: msg:='Invalid slave address';
    16#424A: msg:='Coupling velocity invalid';
    16#424B: msg:='Coupling velocities not constant';
    16#424C: msg:='Cycle time less than or equal to 0.0 not allowed';
    16#424D: msg:='Decoupling task not allowed';
    16#424E: msg:='Function not allowed';
    16#424F: msg:='No valid table weighting has been set';
    16#4250: msg:='Axis type, actual position type or end position type not allowed';
    16#4251: msg:='Function not presently supported';
    16#4252: msg:='State of state machine invalid';
    16#4253: msg:='Reference cam became free too soon';
    16#4254: msg:='Clearance monitoring hardware latch error';
    16#4255: msg:='No memory available';
    16#4256: msg:='Table slave axis has no active table';
    16#4257: msg:='Function not allowed';
    16#4258: msg:='Stopping compensation not allowed';
    16#4259: msg:='Slave table is being used';
    16#425A: msg:='Master or slave axis is processing a job while coupling requested';
    16#425B: msg:='Slave parameter is incorrect';
    16#425C: msg:='Slave type is incorrect';
    16#425D: msg:='Axis stop is already active';
    16#425E: msg:='Maximum number of tables per slave generator reached';
    16#425F: msg:='Scaling mode is invalid';
    16#4260: msg:='Drive disabled';
    16#4261: msg:='Table not found';
    16#4262: msg:='Incorrect table type';
    16#4263: msg:='Single step mode';
    16#4264: msg:='Group task unknown';
    16#4265: msg:='Group function unknown';
    16#4266: msg:='Group task for slave not allowed';
    16#4267: msg:='Group function for slave not allowed';
    16#4268: msg:='NCI Setpoint Generator is Inactive';
    16#4269: msg:='Startposition=Setpoint Position';
    16#426A: msg:='Parameters of delay-generator are invalid';
    16#426B: msg:='External parameters of superimposed instruction invalid';
    16#426C: msg:='Invalid override type';
    16#426D: msg:='Activation position under/overrun';
    16#426E: msg:='Activation impossible: Master is standing';
    16#426F: msg:='Activation mode not possible';
    16#4270: msg:='Start parameter for compensation is invalid';
    16#4271: msg:='Velocity camber is negative';
    16#4272: msg:='Compensation section not positive';
    16#4273: msg:='Target position under/overrun';
    16#4274: msg:='Target position will be under/overrun';
    16#4275: msg:='Group Parameter is Invalid';
    16#4276: msg:='Joint Error at Start of Setpoint Generation';
    16#4277: msg:='Dynamic parameters not permitted';
    16#4279: msg:='New Target Position is Invalid or Cannot be Reached';
    16#427A: msg:='New Velocity for Moving or Final Target Velocity is Invalid';
    16#427B: msg:='Final Velocity or New Target Position is Invalid';
    16#427C: msg:='New Moving Velocity is Invalid';
    16#427D: msg:='Internal Starting Mode is Invalid';
    16#427E: msg:='Motion command could not be realized (BISECTION)';
    16#427F: msg:='New target position has been overrun or will be overrun';
    16#4280: msg:='Group not ready for new task';
    16#4281: msg:='Parameters of oriented stop not admitted';
    16#4282: msg:='Modulo target position of modulo-start is invalid';
    16#4283: msg:='Online change activation mode is invalid';
    16#4284: msg:='Parameterized jerk rate is not permitted';
    16#4285: msg:='Parameterized acceleration or deceleration is not permitted';
    16#4286: msg:='Parameterized velocity is not permitted';
    16#4287: msg:='Activation cannot be executed due to pending activation';
    16#4288: msg:='Illegal combination of different cycle times within axis group';
    16#4289: msg:='Illegal motion reversal';
    16#428A: msg:='Illegal moment for axis command with activation position active';
    16#428B: msg:='Error in stop-calculation routine';
    16#428C: msg:='Command with activation position cannot be performed (path too short)';
    16#428D: msg:='Illegal decouple type when decoupling slave axis';
    16#428E: msg:='Illegal target velocity when decoupling slave axis';
    16#428F: msg:='Command new dynamic parameter requires new target velocity';
    16#4290: msg:='Command with activation position cannot be performed (already in brake phase)';
    16#4291: msg:='Decouple routine of slave axis does not return valid solution';
    16#4292: msg:='Command rejected because command buffer is full';
    16#4293: msg:='Command rejected due to internal error in Look Ahead';
    16#4294: msg:='Command rejected because segment target velocity not realized';
    16#4295: msg:='Successive commands have same final position';
    16#4296: msg:='Logical positioning direction inconsistent with buffer command';
    16#4297: msg:='Command rejected because remaining positioning length too small';
    16#429A: msg:='Restart has Failed';
    16#429B: msg:='Collect error for invalid start parameters';
    16#429C: msg:='Reference cam is not found';
    16#429D: msg:='Reference cam became not free';
    16#429E: msg:='IO sync pulse was not found (hardware latch)';
    16#429F: msg:='Buffer Mode Unknown or not Supported';
    16#42A0: msg:='Coupled axis error';
    16#42A1: msg:='Velocity reduction factor for C0/C1 transition not allowed';
    16#42A2: msg:='Critical angle at segment transition not allowed';
    16#42A3: msg:='Radius of tolerance sphere invalid';
    16#42A5: msg:='Start type invalid';
    16#42A7: msg:='Blending with given parameters not possible';
    16#42A9: msg:='Curve velocity reduction method not allowed';
    16#42AA: msg:='Minimum velocity not allowed';
    16#42AB: msg:='Power function input not allowed';
    16#42AC: msg:='Dynamic change parameter not allowed';
    16#42AD: msg:='Memory allocation error';
    16#42AE: msg:='Calculated end position differs from NC instruction';
    16#42AF: msg:='Calculate remaining chord length invalid';
    16#42B0: msg:='Set value generator SVB active';
    16#42B1: msg:='SVB parameter not allowed';
    16#42B2: msg:='Velocity reduction factor not allowed';
    16#42B3: msg:='Helix is a circle';
    16#42B4: msg:='Helix is a straight line';
    16#42B5: msg:='Guider parameter not allowed';
    16#42B6: msg:='Invalid segment address';
    16#42B7: msg:='Unparameterized generator';
    16#42B8: msg:='Unparameterized table';
    16#42BA: msg:='Calculation of arc length of smoothed path failed';
    16#42BB: msg:='Radius of tolerance ball too small';
    16#42BC: msg:='Error while calculating DXD-Software-Limit switches';
    16#42BD: msg:='NC-Block violates software limit switches of group';
    16#42BE: msg:='Internal error evaluating software limit switch violation';
    16#42BF: msg:='Invalid reference speed type';
    16#42C0: msg:='Interpolating group contains axes of incorrect axis type';
    16#42C1: msg:='Scalar product cannot be calculated';
    16#42C2: msg:='Inverse cosine cannot be calculated';
    16#42C3: msg:='Invalid table entry type';
    16#42C4: msg:='Invalid DIN66025 information type';
    16#42C5: msg:='Invalid dimension';
    16#42C6: msg:='Geometrical object is not a straight line';
    16#42C7: msg:='Geometrical object is not a circle';
    16#42C8: msg:='Geometrical object is not a helix';
    16#42C9: msg:='Set velocity less than or equal to 0.0 is invalid';
    16#42CA: msg:='Address for look-ahead invalid';
    16#42CB: msg:='Set value generator SAF active';
    16#42CC: msg:='CNC set value generation not active';
    16#42CD: msg:='CNC set value generation in stop phase';
    16#42CE: msg:='Override not allowed';
    16#42CF: msg:='Invalid table address';
    16#42D0: msg:='Invalid table entry type';
    16#42D1: msg:='Memory allocation failed (table)';
    16#42D2: msg:='Memory allocation failed (filter)';
    16#42D3: msg:='Filter parameter not allowed';
    16#42D4: msg:='Delete Distance To Go failed';
    16#42D5: msg:='Setpoint generator of flying saw generates incompatible values';
    16#42D6: msg:='Axis stopped to prevent target position overrun';
    16#42D7: msg:='Internal error in transformation from slave to master';
    16#42D8: msg:='Wrong direction in transformation of slave to master';
    16#42DA: msg:='Parameter of Motion Function table incorrect';
    16#42DB: msg:='Motion Function active point references passive point';
    16#42DC: msg:='Internal error by using Motion Function';
    16#42DD: msg:='Axis coupling with synchronization generator declined (incorrect dynamics)';
    16#42DE: msg:='Coupling conditions of synchronization generator incorrect';
    16#42DF: msg:='Moving profile of synchronization generator exceeds dynamic limits';
    16#42E0: msg:='Encoder generator parameter not allowed';
    16#42E1: msg:='External (Fifo) generator parameter not allowed';
    16#42E2: msg:='External generator is active';
    16#42E3: msg:='External generator is not active';
    16#42E4: msg:='NC-Block with auxiliary axis violates software limit switches';
    16#42E5: msg:='NC-Block type Bezier spline curve contains a cusp';
    16#42E7: msg:='Value for dead time compensation not allowed';
    16#42E8: msg:='GROUPERR_RANGE_NOMOTIONWINDOW';
    16#42E9: msg:='GROUPERR_RANGE_NOMOTIONFILTERTIME';
    16#42EA: msg:='GROUPERR_RANGE_TIMEUNITFIFO';
    16#42EB: msg:='GROUPERR_RANGE_OVERRIDETYPE';
    16#42EC: msg:='GROUPERR_RANGE_OVERRIDECHANGETIME';
    16#42ED: msg:='GROUPERR_FIFO_INVALIDDIMENSION';
    16#42EE: msg:='GROUPERR_ADDR_FIFOTABLE';
    16#42EF: msg:='Axis locked for motion commands (stop command active)';
    16#42F0: msg:='Invalid number of auxiliary axes';
    16#42F1: msg:='Invalid reduction parameter for auxiliary axes';
    16#42F2: msg:='Invalid dynamic parameter for auxiliary axes';
    16#42F3: msg:='Invalid coupling parameter for auxiliary axes';
    16#42F4: msg:='Invalid auxiliary axis entry';
    16#42F6: msg:='Invalid limit for velocity reduction of auxiliary axes';
    16#42F8: msg:='Block search: segment not found';
    16#42F9: msg:='Block search: invalid remaining segment length';
    16#42FB: msg:='Internal Error in Context of Coupled Axes';
    16#42FC: msg:='Parameter for Maximum Number of Jobs Invalid';
    16#42FF: msg:='Customer Specific Error';

    // Axis Errors
    16#4300: msg:='Axis ID not allowed';
    16#4301: msg:='Axis type not allowed';
    16#4306: msg:='Slow manual velocity not allowed';
    16#4307: msg:='Fast manual velocity not allowed';
    16#4308: msg:='High speed not allowed';
    16#4309: msg:='Acceleration not allowed';
    16#430A: msg:='Deceleration not allowed';
    16#430B: msg:='Jerk not allowed';
    16#430C: msg:='Delay time between position and velocity not allowed';
    16#430D: msg:='Override type not allowed';
    16#430E: msg:='NCI: Velo-Jump-Factor not allowed';
    16#430F: msg:='NCI: Size of tolerance sphere for auxiliary axis invalid';
    16#4310: msg:='NCI: Maximum deviation for auxiliary axis invalid';
    16#4312: msg:='Referencing velocity in direction of cam not allowed';
    16#4313: msg:='Referencing velocity in sync direction not allowed';
    16#4314: msg:='Pulse width in positive direction not allowed';
    16#4315: msg:='Pulse width in negative direction not allowed';
    16#4316: msg:='Pulse time in positive direction not allowed';
    16#4317: msg:='Pulse time in negative direction not allowed';
    16#4318: msg:='Creep distance in positive direction not allowed';
    16#4319: msg:='Creep distance in negative direction not allowed';
    16#431A: msg:='Braking distance in positive direction not allowed';
    16#431B: msg:='Braking distance in negative direction not allowed';
    16#431C: msg:='Braking time in positive direction not allowed';
    16#431D: msg:='Braking time in negative direction not allowed';
    16#431E: msg:='Switching time from high to low speed not allowed';
    16#431F: msg:='Creep distance for stop not allowed';
    16#4320: msg:='Motion monitoring time not allowed';
    16#4321: msg:='Position window monitoring not allowed';
    16#4322: msg:='Target window monitoring not allowed';
    16#4323: msg:='Loop not allowed';
    16#4324: msg:='Motion monitoring time not allowed';
    16#4325: msg:='Target window range not allowed';
    16#4326: msg:='Position window range not allowed';
    16#4327: msg:='Position window monitoring time not allowed';
    16#4328: msg:='Loop movement not allowed';
    16#4329: msg:='Axis cycle time not allowed';
    16#432A: msg:='Stepper motor operating mode not allowed';
    16#432B: msg:='Displacement per stepper motor step not allowed';
    16#432C: msg:='Minimum speed for stepper motor set value profile not allowed';
    16#432D: msg:='Stepper motor steps per speed level not allowed';
    16#432E: msg:='DWORD for interpretation of axis units not allowed';
    16#432F: msg:='Maximum velocity not allowed';
    16#4330: msg:='Motion monitoring window not allowed';
    16#4331: msg:='PEH time monitoring not allowed';
    16#4332: msg:='PEH monitoring time not allowed';
    16#4333: msg:='Parameter Brake Release Delay is invalid';
    16#4334: msg:='Parameter NC Data Persistence is invalid';
    16#4335: msg:='Parameter for Error Reaction Mode is invalid';
    16#4336: msg:='Parameter for Error Reaction Delay is invalid';
    16#4337: msg:='Parameter Use actual values in deactivated state is invalid';
    16#4338: msg:='Parameter Allow Motion Commands for Slave Axes is invalid';
    16#4339: msg:='Parameter Allow Motion Commands for axis in ext sp gen is invalid';
    16#433A: msg:='Parameter Fading Acceleration is invalid';
    16#433B: msg:='Fast Axis Stop signal type not allowed';
    16#4340: msg:='Axis initialization';
    16#4341: msg:='Group address invalid';
    16#4342: msg:='Encoder address invalid';
    16#4343: msg:='Controller address invalid';
    16#4344: msg:='Drive address invalid';
    16#4345: msg:='Axis interface PLC to NC address invalid';
    16#4346: msg:='Axis interface NC to PLC address invalid';
    16#4347: msg:='Size of axis interface NC to PLC not allowed';
    16#4348: msg:='Size of axis interface PLC to NC not allowed';
    16#4356: msg:='Controller enable';
    16#4357: msg:='Negative limit hit';
    16#4358: msg:='Positive limit hit';
    16#4359: msg:='Set velocity not allowed';
    16#435A: msg:='Movement smaller than one encoder increment';
    16#435B: msg:='Set acceleration monitoring';
    16#435C: msg:='PEH time monitoring';
    16#435D: msg:='Motion Monitoring';
    16#435E: msg:='Looping distance less than breaking distance';
    16#435F: msg:='Starting velocity not allowed';
    16#4360: msg:='Final velocity not allowed';
    16#4361: msg:='Time range exceeded (future)';
    16#4362: msg:='Time range exceeded (past)';
    16#4363: msg:='Position cannot be determined';
    16#4364: msg:='Position indeterminable (conflicting direction of travel)';
    16#4370: msg:='No slave coupling possible (velocity violation)';
    16#4371: msg:='No slave coupling possible (acceleration violation)';
    16#43A0: msg:='Axis consequential error';

    // Encoder Errors
    16#4400: msg:='Encoder ID not allowed';
    16#4401: msg:='Encoder type not allowed';
    16#4402: msg:='Encoder mode not allowed';
    16#4403: msg:='Encoder counting direction inverted?';
    16#4404: msg:='Referencing status';
    16#4405: msg:='Encoder increments for each physical rotation invalid';
    16#4406: msg:='Scaling factor not allowed';
    16#4407: msg:='Position offset (zero point offset) not allowed';
    16#4408: msg:='Modulo factor not allowed';
    16#4409: msg:='Position filter time not allowed';
    16#440A: msg:='Velocity filter time not allowed';
    16#440B: msg:='Acceleration filter time not allowed';
    16#440C: msg:='Cycle time not allowed';
    16#440D: msg:='Configuration of selected units is invalid';
    16#440E: msg:='Actual position correction / measurement system error correction not allowed';
    16#440F: msg:='Filter time actual position correction not allowed';
    16#4410: msg:='Search direction for referencing cam inverted';
    16#4411: msg:='Search direction for sync pulse inverted';
    16#4412: msg:='Reference position not allowed';
    16#4413: msg:='Clearance monitoring between hardware latch and sync pulse not allowed';
    16#4414: msg:='Minimum clearance between hardware latch and sync pulse not allowed';
    16#4415: msg:='External sync pulse not allowed';
    16#4416: msg:='Scaling of noise rate is not allowed';
    16#4417: msg:='Tolerance window for modulo-start invalid';
    16#4418: msg:='Encoder reference mode not allowed';
    16#4419: msg:='Encoder evaluation direction not allowed';
    16#441A: msg:='Encoder reference system invalid';
    16#441B: msg:='Encoder position initialization mode invalid';
    16#441C: msg:='Encoder sign interpretation invalid';
    16#441D: msg:='Homing Sensor Source invalid';
    16#4420: msg:='Software end location monitoring minimum not allowed';
    16#4421: msg:='Software end location monitoring maximum not allowed';
    16#4422: msg:='Actual value setting is outside the value range';
    16#4423: msg:='Software end location minimum not allowed';
    16#4424: msg:='Software end location maximum not allowed';
    16#4425: msg:='Filter mask for raw data of encoder is invalid';
    16#4426: msg:='Reference mask for raw data of encoder is invalid';
    16#4427: msg:='Parameter Dead Time Compensation Mode (Encoder) is Invalid';
    16#4428: msg:='Parameter Control Bits of Dead Time Compensation (Encoder) is Invalid';
    16#4429: msg:='Parameter Time Related Shift of Dead Time Compensation Mode (Encoder) is Invalid';
    16#4430: msg:='Hardware latch activation (encoder)';
    16#4431: msg:='External hardware latch activation (encoder)';
    16#4432: msg:='External hardware latch activation (encoder) - latch valid';
    16#4433: msg:='External hardware latch activation (encoder) - handshake active';
    16#4434: msg:='Encoder function not supported';
    16#4435: msg:='Encoder function is already active';
    16#4440: msg:='Encoder initialization';
    16#4441: msg:='Axis address invalid';
    16#4442: msg:='I/O input structure address invalid';
    16#4443: msg:='I/O output structure address invalid';
    16#4450: msg:='Encoder counter underflow monitoring';
    16#4451: msg:='Encoder counter overflow monitoring';
    16#4460: msg:='Minimum Software Position Limit (Axis Start)';
    16#4461: msg:='Maximum Software Position Limit (Axis Start)';
    16#4462: msg:='Minimum Software Position Limit (Positioning Process)';
    16#4463: msg:='Maximum Software Position Limit (Positioning Process)';
    16#4464: msg:='Encoder hardware error';
    16#4465: msg:='Position initialization error at system start';
    16#4466: msg:='Invalid I/O data for more than n continuous NC cycles (encoder)';
    16#4467: msg:='Encoder error: invalid actual position data';
    16#4468: msg:='Invalid IO Input Data (Error Type 1)';
    16#4469: msg:='Invalid IO Input Data (Error Type 2)';
    16#4470: msg:='SSI transformation fault or not finished';
    16#44A2: msg:='ENCERR_ADDR_CONTROLLER';
    16#44A3: msg:='ENCERR_INVALID_CONTROLLERTYPE';

    // Controller Errors
    16#4500: msg:='Controller ID not allowed';
    16#4501: msg:='Controller type not allowed';
    16#4502: msg:='Controller operating mode not allowed';
    16#4503: msg:='Weighting of velocity pre-control not allowed';
    16#4504: msg:='Following error monitoring (position) not allowed';
    16#4505: msg:='Following error (velocity) not allowed';
    16#4506: msg:='Following error window (position) not allowed';
    16#4507: msg:='Following error filter time (position) not allowed';
    16#4508: msg:='Following error window (velocity) not allowed';
    16#4509: msg:='Following error filter time (velocity) not allowed';
    16#450A: msg:='Controller Output Limitation Improper';
    16#4510: msg:='Proportional gain Kv or Kp (controller) not allowed';
    16#4511: msg:='Integral-action time Tn (controller) not allowed';
    16#4512: msg:='Derivative action time Tv (controller) not allowed';
    16#4513: msg:='Damping time Td (controller) not allowed';
    16#4514: msg:='Activation of automatic offset compensation not allowed';
    16#4515: msg:='Additional proportional gain Kv or Kp (controller) not allowed';
    16#4516: msg:='Reference velocity for additional proportional gain not allowed';
    16#4517: msg:='Proportional gain Pa (proportion) not allowed';
    16#4518: msg:='Proportional gain Kv (velocity controller) not allowed';
    16#4519: msg:='Reset time Tn (velocity controller) not allowed';
    16#451C: msg:='Velocity Filter Time Improper';
    16#451D: msg:='Dead zone not allowed';
    16#451F: msg:='Proportionality Factor Kcp Improper';
    16#4520: msg:='Rate time Tv (velocity controller) not allowed';
    16#4521: msg:='Damping time Td (velocity controller) not allowed';
    16#4522: msg:='Limitation of the I Part Improper';
    16#4523: msg:='Limitation of the D Part Improper';
    16#4524: msg:='Parameter Switching Off the I Part During Motion is Improper';
    16#4525: msg:='Parameter Filter Time for P-T2 Filter Improper';
    16#4526: msg:='Velocity Observer: Parameterized Mode is Improper';
    16#4527: msg:='Velocity Observer: Motor Torque Constant Kt or Kf is Improper';
    16#4528: msg:='Velocity Observer: Motor Moment of Inertia JM is Improper';
    16#4529: msg:='Velocity Observer: Band Width f0 is Improper';
    16#452A: msg:='Velocity Observer: Correction Factor kc is Improper';
    16#452B: msg:='Velocity Observer: Time Constant T for First Order Filter is Improper';
    16#452C: msg:='Velocity Observer: Amplitude Damping d for Second Order Filter is Improper';
    16#452D: msg:='Velocity Observer: Frequency fHP or fTP for Second Order Filter is Improper';
    16#4540: msg:='Controller initialization';
    16#4541: msg:='Axis address invalid';
    16#4542: msg:='Drive address invalid';
    16#4550: msg:='Stall: position lag monitoring error';
    16#4551: msg:='Following error monitoring (velocity)';
    16#45A0: msg:='CONTROLERR_RANGE_AREA_ASIDE';
    16#45A1: msg:='CONTROLERR_RANGE_AREA_BSIDE';
    16#45A2: msg:='CONTROLERR_RANGE_QNENN';
    16#45A3: msg:='CONTROLERR_RANGE_PNENN';
    16#45A4: msg:='CONTROLERR_RANGE_AXISIDPRESP0';

    // Drive Errors
    16#4600: msg:='Drive ID not allowed';
    16#4601: msg:='Drive type impermissible';
    16#4602: msg:='Drive operating mode impermissible';
    16#4603: msg:='Motor polarity inverted?';
    16#4604: msg:='Drift compensation/speed offset (DAC offset)';
    16#4605: msg:='Reference speed (velocity pre-control)';
    16#4606: msg:='Reference output in percent';
    16#4607: msg:='Quadrant compensation factor';
    16#4608: msg:='Velocity reference point';
    16#4609: msg:='Output reference point';
    16#460A: msg:='Minimum or maximum output limits (output limitation)';
    16#460B: msg:='DRIVEERR_RANGE_MAXINCREMENT';
    16#460C: msg:='DRIVEERR_RANGE_DRIVECONTROLDWORD';
    16#460D: msg:='DRIVEERR_RANGE_RESETCYCLECOUNTER';
    16#460F: msg:='Drive torque output scaling impermissible';
    16#4610: msg:='Drive velocity output scaling is not allowed';
    16#4611: msg:='Profi Drive DSC proportional gain Kpc (controller) impermissible';
    16#4612: msg:='Table ID is impermissible';
    16#4613: msg:='Table interpolation type is impermissible';
    16#4614: msg:='Output offset in percent is impermissible';
    16#4615: msg:='Profi Drive DSC scaling for calculation of Xerr (controller) impermissible';
    16#4616: msg:='Drive acceleration output scaling impermissible';
    16#4617: msg:='Drive position output scaling impermissible';
    16#461C: msg:='Drive filter type impermissible for command variable filter';
    16#461D: msg:='Drive filter time impermissible for command variable filter';
    16#461E: msg:='Drive filter order impermissible for command variable filter';
    16#4620: msg:='Bit mask for stepper motor cycle impermissible';
    16#4621: msg:='Bit mask for stepper motor holding current impermissible';
    16#4622: msg:='Scaling factor for actual torque (actual current) impermissible';
    16#4623: msg:='Filter time for actual torque is impermissible';
    16#4624: msg:='Filter time for temporal derivation of actual torque is impermissible';
    16#4627: msg:='DRIVEOPERATIONMODEBUSY';
    16#4630: msg:='Overtemperature';
    16#4631: msg:='Undervoltage';
    16#4632: msg:='Wire break in phase A';
    16#4633: msg:='Wire break in phase B';
    16#4634: msg:='Overcurrent in phase A';
    16#4635: msg:='Overcurrent in phase B';
    16#4636: msg:='Torque overload (stall)';
    16#4640: msg:='Drive initialization';
    16#4641: msg:='Axis address invalid';
    16#4642: msg:='Address IO input structure invalid';
    16#4643: msg:='Address IO output structure invalid';
    16#4650: msg:='Drive hardware not ready to operate';
    16#4651: msg:='Error in cyclic communication of drive (Life Counter)';
    16#4652: msg:='Changing table ID when active controller enable is impermissible';
    16#4655: msg:='Invalid IO data';

    // NC-PLC Errors
    16#4B00: msg:='Axis was stopped';
    16#4B01: msg:='Axis cannot be started';
    16#4B02: msg:='Control mode not permitted';
    16#4B03: msg:='Axis is not moving';
    16#4B04: msg:='Invalid mode';
    16#4B05: msg:='Command not permitted';
    16#4B06: msg:='Parameter incorrect';
    16#4B07: msg:='Timeout axis function block after 6 seconds';
    16#4B08: msg:='Axis is in protected mode';
    16#4B09: msg:='Axis is not ready';
    16#4B0A: msg:='Error during referencing';
    16#4B0B: msg:='Incorrect definition of trigger input';
    16#4B0C: msg:='Position latch was disabled';
    16#4B0D: msg:='NC status feedback timeout';
    16#4B0E: msg:='Additional product not installed';
    16#4B0F: msg:='No NC Cycle Counter Update';
    16#4B10: msg:='M-function query missing';
    16#4B11: msg:='Zero shift index is outside the range';
    16#4B12: msg:='R-parameter index or size is invalid';
    16#4B13: msg:='Index for tool description is invalid';
    16#4B14: msg:='Version of cyclic channel interface does not match';
    16#4B15: msg:='Channel is not ready for requested function';
    16#4B16: msg:='Requested function is not activated';
    16#4B17: msg:='Axis is already in another group';
    16#4B18: msg:='Block search could not be executed successfully';
    16#4B19: msg:='Invalid block search parameter';
    16#4B20: msg:='Cannot add all axes';
    16#4B30: msg:='Pointer is invalid';
    16#4B31: msg:='Memory size invalid';
    16#4B32: msg:='Cam table ID is invalid';
    16#4B33: msg:='Point ID is invalid';
    16#4B34: msg:='Number of points is invalid';
    16#4B35: msg:='MC table type is invalid';
    16#4B36: msg:='Number of rows invalid';
    16#4B37: msg:='Number of columns invalid';
    16#4B38: msg:='Step size invalid';
    16#4B40: msg:='Terminal type not supported';
    16#4B41: msg:='Register read/write error';
    16#4B42: msg:='Axis is enabled';
    16#4B43: msg:='Incorrect size of compensation table';
    16#4B44: msg:='Min/max position in compensation table does not match';
    16#4B45: msg:='Not implemented';
    16#4B46: msg:='Window not in specified modulo range';
    16#4B47: msg:='Buffer overflow';
    16#4B60: msg:='Motion command did not become active';
    16#4B61: msg:='Motion command could not be monitored by PLC';
    16#4B62: msg:='Buffered command was terminated with an error';
    16#4B63: msg:='Buffered command was completed without feedback';
    16#4B64: msg:='BufferMode is not supported by command';
    16#4B65: msg:='Command number is zero';
    16#4B66: msg:='Function block was not called cyclically';
    16#4B71: msg:='Invalid NCI entry type';
    16#4B72: msg:='NCI feed table full';
    16#4B73: msg:='Internal error';
    16#4B74: msg:='ST_NciTangentialFollowingDesc: Tangential axis is not auxiliary axis';
    16#4B75: msg:='ST_NciTangentialFollowingDesc: nPathAxis1 or nPathAxis2 is not path axis';
    16#4B76: msg:='ST_NciTangentialFollowingDesc: nPathAxis1 and nPathAxis2 are the same';
    16#4B77: msg:='ST_NciGeoCirclePlane: Circle incorrectly parameterized';
    16#4B78: msg:='Internal error during calculation of tangential following';
    16#4B79: msg:='Tangential following: Monitoring of deviation angle detected large deviation';
    16#4B7A: msg:='Not implemented';
    16#4B7B: msg:='Tangential following: radius of current arc is too small';
    16#4B7C: msg:='FB_NciFeedTablePreparation: pEntry is NULL';
    16#4B7D: msg:='FB_NciFeedTablePreparation: specified nEntryType does not match structure type';
    16#4B7E: msg:='ST_NciMFuncFast and ST_NciMFuncHsk: M-function not between 0 and 159';
    16#4B7F: msg:='ST_NciDynOvr: requested value for dynamic override not between 0.01 and 1';
    16#4B80: msg:='ST_NciVertexSmoothing: invalid parameter';
    16#4B81: msg:='FB_NciFeedTablePreparation: requested velocity not in valid range';
    16#4B82: msg:='ST_Nci*: invalid parameter';
    16#4B90: msg:='Determined drive type is not supported';
    16#4B91: msg:='Direction is impermissible';
    16#4B92: msg:='SwitchMode is impermissible';
    16#4B93: msg:='Mode for parameter handling is impermissible';
    16#4B94: msg:='Parameterization of torque limits is inconsistent';
    16#4B95: msg:='Parameterization of position lag limit is impermissible';
    16#4B96: msg:='Parameterization of distance limit is impermissible';
    16#4B97: msg:='Attempt to back up parameters again (already backed up)';
    16#4B98: msg:='Attempt to restore parameters (none have been backed up)';
    16#4B9F: msg:='Abortion of homing has failed';
    16#4BA0: msg:='KinGroup error: kinematic group is in error state';
    16#4BA1: msg:='KinGroup timeout: timeout during call of kinematic block';
    16#4BB0: msg:='Current axis position or position with new offset exceeds valid range';
    16#4BB1: msg:='New position offset exceeds valid range';
    16#4BB2: msg:='Current axis position or position with new offset below valid range';
    16#4BB3: msg:='New position offset falls below valid range';
    16#4BB4: msg:='Activated feedback and/or storage location differ from parameterization';
    16#4BB5: msg:='Reinitialization of actual NC position has failed';
    16#4BB6: msg:='Command to set or delete position offset rejected without feedback';
    16#4BB7: msg:='Command to set or delete position offset rejected with feedback';
    16#4BB8: msg:='Firmware version >= 19 required for servo terminal';
    16#4BB9: msg:='Modulo settings on drive controller and NC are different';
    16#4BC2: msg:='New position offset exceeds valid value range';
    16#4BC3: msg:='I/O data are invalid or terminal is in error state';
    16#4FFF: msg:='Unknown NC error (not in manual)';

    // Custom error definitions
    E_LCLSMotionError.ABORTED: msg:='Aborted move request with active move in progress';
    E_LCLSMotionError.UNSAFE: msg:='Position state unsafe';
    E_LCLSMotionError.INVALID: msg:='Position state invalid';
    E_LCLSMotionError.TEST: msg:='Fake testing error';

    // Fallbacks
    0: msg:='';
    ELSE
        msg:='Contact PCDS to add new message';
END_CASE
F_MotionErrorCodeLookup := msg;

END_FUNCTION

// ---- Tests/Helpers/FB_TestHelperSetAndMove.TcPOU
FUNCTION_BLOCK FB_TestHelperSetAndMove
(*
    Set an stMotionStage to a start position, then cause a move.
    On rising edge of bExecute, errors are cleared, the user enable is set to FALSE, and the position is set.
    After the position is set, user enable is re-introduced and a move begins.

    The progress of this function block for the purposes of a unit test can be monitored via the outputs.

    The motion stage should have its own FB_MotionStage or some stand-in for it running on outside of the FB.

    This is, in itself, tested in FB_TestHelperSetAndMove_Test.
*)
VAR_IN_OUT
    // The motion state to test with
    stMotionStage: ST_MotionStage;
END_VAR
VAR_INPUT
    // Begin on rising edge, stop on falling edge.
    bExecute: BOOL;
    // The position to set the motor to
    fStartPosition: LREAL;
    // The goal to move the motor towards
    fGoalPosition: LREAL;
    // The velocity to move at
    fVelocity: LREAL;
    // If TRUE, we'll set all the hardware enable signals. Leave this as FALSE if your testing involves any of the hardware enables.
    bHWEnable: BOOL;
END_VAR
VAR_OUTPUT
    // Goes to TRUE once the motor has no errors and is deactivated.
    bResetDone: BOOL;
    // Goes to TRUE once the set position completes.
    bSetDone: BOOL;
    // Goes to TRUE once the motor begins moving.
    bMotionStarted: BOOL;
    // Goes to TRUE once the motor reaches its destination.
    bMoveDone: BOOL;
    // If bBusy is FALSE, the function block is ready for a new request. Goes to TRUE after bExecute rises and back to FALSE after bMoveDone or bError rises. Also goes to FALSE after the motor stops following bExecute being dropped to FALSE.
    bBusy: BOOL;
    // Goes to TRUE in case of an error from FB_MotionRequest
    bError: BOOL;
    // Counts up from bExecute's rising trigger. Can be used to implement a timeout.
    tElapsed: TIME;
    // Current motor position in case you're looking for it
    fActPosition: LREAL;
    // Goes to TRUE if we're trying to stop a move. We'll stop an in-progress move when bExecute goes to FALSE, and we'll make sure the motor fully stops before responding to the next bExecute rising edge.
    bStoppingMotor: BOOL;
END_VAR
VAR
    fbMoveRequest: FB_MotionRequest;
    mcSetPos: MC_SetPosition;
    tonTimeout: TON;
    rtExec: R_TRIG;
    ftExec: F_TRIG;
    bExecQueued: BOOL;
    nLatchError: UDINT;
END_VAR


tonTimeout(
    IN:=bExecute,
    PT:=T#1h,
    ET=>tElapsed,
);
rtExec(CLK:=bExecute);
ftExec(CLK:=bExecute);

// Set the outputs to known values on exec
bResetDone R= rtExec.Q;
bSetDone R= rtExec.Q;
bMotionStarted R= rtExec.Q;
bMoveDone R= rtExec.Q;
bBusy S= rtExec.Q;
bError R= rtExec.Q;

bExecQueued S= rtExec.Q;
bExecQueued R= ftExec.Q;
bStoppingMotor S= ftExec.Q;

// Set the hardware enables if asked
IF bHWEnable THEN
    stMotionStage.bLimitForwardEnable := TRUE;
    stMotionStage.bLimitBackwardEnable := TRUE;
    stMotionStage.bHardwareEnable := TRUE;
    stMotionStage.bPowerSelf := TRUE;
END_IF


// Note that we only reset if it's needed, e.g. the motor has an error or is enabled or moving etc. etc.
bResetDone S= stMotionStage.bError = FALSE AND stMotionStage.bBusy = FALSE AND stMotionStage.bAllEnable = FALSE;

// All uses of fbMoveRequest are in this IF/ELSE tree
IF bStoppingMotor THEN
    // Continue stopping the motor from previous cycles
    fbMoveRequest(
        stMotionStage:=stMotionStage,
        bExecute:=FALSE,
    );
    stMotionStage.bExecute := FALSE;
    bStoppingMotor R= NOT stMotionStage.Axis.Status.ControlLoopClosed AND NOT fbMoveRequest.bBusy;
ELSIF bExecQueued THEN
    // First exec cycle: bring these to FALSE for later use
    bExecQueued := FALSE;
    stMotionStage.bUserEnable := FALSE;
    fbMoveRequest(
        stMotionStage:=stMotionStage,
        bExecute:=FALSE,
        bReset:=FALSE,
    );
ELSIF NOT bResetDone THEN
    // Other cycles: reset until we're done resetting
    fbMoveRequest(
        stMotionStage:=stMotionStage,
        bReset:=bExecute,
    );
ELSIF fStartPosition <> fGoalPosition THEN
    // Later: do the move
    // Important to not enable the motor until the set position is done
    stMotionStage.bUserEnable := bSetDone;
    fbMoveRequest(
        stMotionStage:=stMotionStage,
        bExecute:=bSetDone AND bExecute AND NOT bMoveDone AND NOT bError,
        bReset:=FALSE,
        enumMotionRequest:=E_MotionRequest.INTERRUPT,
        fPos:=fGoalPosition,
        fVel:=fVelocity,
    );
    bMotionStarted S= bSetDone AND fbMoveRequest.bExecute AND stMotionStage.bBusy AND stMotionStage.stAxisStatus.fActPosition <> fStartPosition;
    bMoveDone S= bMotionStarted AND stMotionStage.stAxisStatus.fActPosition = fGoalPosition;
ELSIF fStartPosition = fGoalPosition THEN
    // if the start position matches the goal position, make sure the commanded position is
    // set to the current position.
    stMotionStage.fPosition := fGoalPosition;
END_IF

// Set the position prior to the move but after the reset.
mcSetPos(
    Axis:=stMotionStage.Axis,
    Execute:=bResetDone AND bExecute AND NOT bSetDone AND NOT bError,
    Position:=fStartPosition,
);
IF mcSetPos.Done OR mcSetPos.Error THEN
    nLatchError := mcSetPos.ErrorID;
END_IF
bSetDone S= mcSetPos.Done AND NOT mcSetPos.Error AND stMotionStage.stAxisStatus.fActPosition = fStartPosition;

// Any sub-error is an error here
bError := fbMoveRequest.bError OR mcSetPos.Error;

// Reset bBusy when appropriate
bBusy R= (bMoveDone AND NOT bStoppingMotor) OR bError OR ftExec.Q;

// Extract the motor position
fActPosition := stMotionStage.stAxisStatus.fActPosition;

END_FUNCTION_BLOCK

// ---- POUs/Motion/FB_MotionRequest.TcPOU
FUNCTION_BLOCK FB_MotionRequest
(*
    Request a move from an axis controlled via EPICS using FB_MotionStage
    This exists to manage situations where different bits of code may need to move the same motor.
    With just the ST_MotionStage/FB_MotionStage setup it is possible for two function blocks to
    fight with and interfere with each other and with the EPICS commands.
*)
VAR_IN_OUT
    // Motor to move
    stMotionStage: ST_MotionStage;
END_VAR
VAR_INPUT
    // Start move on rising edge, stop move on falling edge
    bExecute: BOOL;
    // Reset errors on rising edge
    bReset: BOOL;
    // Define behavior for when the motor is already moving
    enumMotionRequest: E_MotionRequest := E_MotionRequest.WAIT;
    // Goal position
    fPos: LREAL;
    // Move velocity
    fVel: LREAL;
    // Optional acceleration
    fAcc: LREAL;
    // Optional deceleration
    fDec: LREAL;
END_VAR
VAR_OUTPUT
    // True if in error state
    bError: BOOL;
    // Error code
    nErrorId: UDINT;
    // What the error code means
    sErrorMessage: STRING;
    // If TRUE, we are moving the motor
    bBusy: BOOL;
    // If TRUE, we are not moving the motor and our most recent move was successful
    bDone: BOOL;
END_VAR
VAR
    rtExec: R_TRIG;
    ftExec: F_TRIG;
    rtReset: R_TRIG;
    ftBusy: F_TRIG;
    nState: UINT := 0;
    bMyMove: BOOL;
    bCausedError: BOOL;
END_VAR
// Define local constants for our state machine states
VAR CONSTANT
    INIT: UINT := 0;
    WAIT_EXEC: UINT := 1;
    PICK_REQUEST: UINT := 2;
    WAIT_OTHER_MOVE: UINT := 3;
    STOP_OTHER_MOVE: UINT := 4;
    START_MOVE: UINT := 5;
    WAIT_MY_MOVE: UINT := 6;
    STOP_MY_MOVE: UINT := 7;
    DONE_MOVING: UINT := 8;
    ERROR: UINT := 9;
END_VAR

rtExec(CLK:=bExecute);
ftExec(CLK:=bExecute);
rtReset(CLK:=bReset);

// Go back to INIT state on reset
IF rtReset.Q THEN
    nState := INIT;
    stMotionStage.bReset := TRUE;
END_IF
IF rtExec.Q OR ftExec.Q THEN
    bDone := FALSE;
END_IF

CASE nState OF
    // Start by setting everything to a known value
    INIT:
        nState := WAIT_EXEC;
        bError := FALSE;
        sErrorMessage := '';
        bDone := FALSE;
        bCausedError := FALSE;
    // Normal "waiting for move command" state
    WAIT_EXEC:
        bMyMove := FALSE;
        // Looking for a rising edge on bExecute
        IF rtExec.Q THEN
            bDone := FALSE;
            nState := PICK_REQUEST;
        END_IF
    // Decide how to handle the request
    PICK_REQUEST:
        IF stMotionStage.bBusy THEN
            CASE enumMotionRequest OF
                E_MotionRequest.WAIT:
                    nState := WAIT_OTHER_MOVE;
                E_MotionRequest.INTERRUPT:
                    nState := STOP_OTHER_MOVE;
                E_MotionRequest.ABORT:
                    nState := ERROR;
                    bError := TRUE;
                    nErrorId := E_LCLSMotionError.ABORTED;
            END_CASE
        ELSE
            nState := START_MOVE;
        END_IF
    // Watch the other move, then see if it's our turn
    WAIT_OTHER_MOVE:
        IF NOT stMotionStage.bBusy THEN
            // Try to pick request again next cycle once the move is over
            nState := PICK_REQUEST;
        END_IF
    // Interrupt the other move, then go to start ours
    STOP_OTHER_MOVE:
        stMotionStage.bExecute := FALSE;
        IF NOT stMotionStage.bBusy THEN
            nState := START_MOVE;
        END_IF
    // Set the correct values on ST_MotionStage to start a new absolute move
    START_MOVE:
        bMyMove := TRUE;
        stMotionStage.bExecute := TRUE;
        stMotionStage.nCommand := E_EpicsMotorCmd.MOVE_ABSOLUTE;
        stMotionStage.fPosition := fPos;
        stMotionStage.fVelocity := fVel;
        stMotionStage.fAcceleration := fAcc;
        stMotionStage.fDeceleration := fDec;
        nState := WAIT_MY_MOVE;
    // Watch our ongoing move, look for the move to end or requests to stop the move from this FB
    WAIT_MY_MOVE:
        ftBusy(CLK:=stMotionStage.bBusy);
        IF ftBusy.Q THEN
            nState := DONE_MOVING;
        END_IF
        // Implement stop on falling trigger
        IF ftExec.Q THEN
            nState := STOP_MY_MOVE;
        END_IF
    // Request a stop and wait for it to happen
    STOP_MY_MOVE:
        stMotionStage.bExecute := FALSE;
        IF NOT stMotionStage.bBusy THEN
            nState := DONE_MOVING;
        END_IF
    // Pick out the bDone state and return to waiting
    DONE_MOVING:
        bDone := stMotionStage.bDone;
        nState := WAIT_EXEC;
    // Lock us into the error state until the FB is reset
    ERROR:
        bMyMove := FALSE;
END_CASE

// Transition to the ERROR state if applicable
IF bMyMove AND stMotionStage.bError THEN
    nState := ERROR;
    bError := TRUE;
    nErrorId := stMotionStage.nErrorId;
    bCausedError := TRUE;
END_IF
sErrorMessage := F_MotionErrorCodeLookup(nErrorId := nErrorId);

CASE nState OF
INIT, WAIT_EXEC, ERROR:
    bBusy := FALSE;
ELSE
    bBusy := TRUE;
END_CASE

END_FUNCTION_BLOCK

// ---- POUs/Motion/States/Internals/FB_PositionStateInternal.TcPOU
FUNCTION_BLOCK FB_PositionStateInternal
(*
    Routines that must be called on all ST_PositionState

    Currently, this FB:
    - ensures that a position state has both a proper encoder count
      and a proper position in engineering units with both of these quantities matching
    - handles the parameter locking feature, which nominally prevents the user from changing
      details about a locked state via EPICS
*)
VAR_IN_OUT
    stMotionStage: ST_MotionStage;
    stPositionState: ST_PositionState;
END_VAR
VAR_OUTPUT
END_VAR
VAR
    fbEncConverter: FB_RawCountConverter;
    fbLock: FB_PositionStateLock;
END_VAR

// Mark that we've been here
stPositionState.bUpdated := TRUE;

// Update pos state's count or egu position as appropriate
IF stMotionStage.bAxisParamsInit THEN
    fbEncConverter(
        stParameters:=stMotionStage.stAxisParameters,
        nCountCheck:=stPositionState.nEncoderCount,
        fPosCheck:=stPositionState.fPosition);
    IF stPositionState.bUseRawCounts THEN
        stPositionState.fPosition := fbEncConverter.fPosGet;
    ELSE
        stPositionState.nEncoderCount := fbEncConverter.nCountGet;
    END_IF
END_IF

// Handle state parameter locking
fbLock(
    stPositionState:=stPositionState,
    bEnable:=stMotionStage.bAxisParamsInit);

END_FUNCTION_BLOCK

// ---- POUs/Motion/States/Helpers/FB_RawCountConverter.TcPOU
FUNCTION_BLOCK FB_RawCountConverter
(*
    Utility function block for converting raw counts to EGU and back
*)
VAR_INPUT
    // Parameters to check against
    stParameters: ST_AxisParameterSet;
    // Optional count to convert to a real position
    nCountCheck: UDINT;
    // Optional position to convert to encoder counts
    fPosCheck: LREAL;
END_VAR
VAR_OUTPUT
    // If converting position, the number of counts
    nCountGet: UDINT;
    // If converting counts, the position
    fPosGet: LREAL;
    // True during a parameter get/calc
    bBusy: BOOL;
    // True after a successful get/calc
    bDone: BOOL;
    // True if the calculation errored
    bError: BOOL;
END_VAR

IF stParameters.fEncScaleFactorInternal <> 0 THEN
    nCountGet := LREAL_TO_UDINT((fPosCheck - stParameters.fEncOffset) / stParameters.fEncScaleFactorInternal);
    fPosGet := nCountCheck * stParameters.fEncScaleFactorInternal + stParameters.fEncOffset;
END_IF

END_FUNCTION_BLOCK

// ---- POUs/Motion/States/Internals/FB_PositionStateLock.TcPOU
FUNCTION_BLOCK FB_PositionStateLock
(*
    Implements immutability for a locked ST_PositionState
    Once this is called the first time, the parameters at the time of the call will be restored on all subsequent calls.
*)
VAR_IN_OUT
    stPositionState: ST_PositionState;
END_VAR
VAR_INPUT
    bEnable: BOOL;
END_VAR
VAR
    stCachedPositionState: ST_PositionState;
    bInit: BOOL := FALSE;
END_VAR

IF bEnable THEN
    // Force values to be cached if we've cached something
    IF bInit AND stPositionState.bLocked THEN
        stPositionState.sName := stCachedPositionState.sName;
        stPositionState.fPosition := stCachedPositionState.fPosition;
        stPositionState.fDelta := stCachedPositionState.fDelta;
        stPositionState.fVelocity := stCachedPositionState.fVelocity;
        stPositionState.fAccel := stCachedPositionState.fAccel;
        stPositionState.fDecel := stCachedPositionState.fDecel;
    // If we haven't cached and we should, make the cache. Note that we skip bLocked, bValid, and bMoveOk
    ELSIF NOT bInit AND stPositionState.bLocked THEN
        stCachedPositionState.sName := stPositionState.sName;
        stCachedPositionState.fPosition := stPositionState.fPosition;
        stCachedPositionState.fDelta := stPositionState.fDelta;
        stCachedPositionState.fVelocity := stPositionState.fVelocity;
        stCachedPositionState.fAccel := stPositionState.fAccel;
        stCachedPositionState.fDecel := stPositionState.fDecel;
        bInit := TRUE;
    // Do nothing, or unlock the state if bLocked goes FALSE
    ELSIF NOT stPositionState.bLocked THEN
        bInit := FALSE;
    END_IF
END_IF

END_FUNCTION_BLOCK

// ---- POUs/Motion/States/Helpers/F_AtPositionState.TcPOU
FUNCTION F_AtPositionState : BOOL
(*
    Check if the motor is within the state bounds
    This will only run properly if FB_PositionStateInternal has been called on the position state to initialize it.
*)
VAR_INPUT
    stMotionStage: ST_MotionStage;
    stPositionState: ST_PositionState;
END_VAR

// If state is defined, we are within the delta, and we are either not moving or our destination is within the delta, we are at the state
F_AtPositionState := stPositionState.bValid AND stPositionState.bUpdated
                     AND F_PosWithinDelta(stMotionStage.stAxisStatus.fActPosition, stPositionState)
                     AND ((NOT stMotionStage.bExecute) OR F_PosWithinDelta(stMotionStage.fPosition, stPositionState));

END_FUNCTION

// ---- POUs/Motion/States/Helpers/F_PosWithinDelta.TcPOU
FUNCTION F_PosWithinDelta : BOOL
VAR_INPUT
    fPosition: LREAL;
    stPositionState: ST_PositionState;
END_VAR

F_PosWithinDelta := F_PosOverLowerBound(fPosition, stPositionState) AND
                    F_PosUnderUpperBound(fPosition, stPositionState);

END_FUNCTION

// ---- POUs/Motion/States/Helpers/F_PosOverLowerBound.TcPOU
FUNCTION F_PosOverLowerBound : BOOL
VAR_INPUT
    fPosition: LREAL;
    stPositionState: ST_PositionState;
END_VAR

F_PosOverLowerBound := fPosition > (stPositionState.fPosition - ABS(stPositionState.fDelta));

END_FUNCTION

// ---- POUs/Motion/States/Helpers/F_PosUnderUpperBound.TcPOU
FUNCTION F_PosUnderUpperBound : BOOL
VAR_INPUT
    fPosition: LREAL;
    stPositionState: ST_PositionState;
END_VAR

F_PosUnderUpperBound := fPosition < (stPositionState.fPosition + ABS(stPositionState.fDelta));

END_FUNCTION

// ---- Tests/FB_AxisParameterSetExposed_Test.TcPOU
FUNCTION_BLOCK FB_AxisParameterSetExposed_Test EXTENDS FB_MotorTestSuite
(*
    Quick Check to verify exposed NC parameters are copied properly.
*)
VAR
    stMotionStage: ST_MotionStage;
    fbMotionStage: FB_MotionStage;
    nTestCounter: UINT;
    bOneTestDone: BOOL;
    tonTimer: TON;
END_VAR

IF nTestCounter = 0 THEN
    nTestCounter := 1;
END_IF

// Test that parameters are copied to the exposed parameters properly.
TestParameterCopy(1);

IF bOneTestDone THEN
    bOneTestDone := FALSE;
    nTestCounter := nTestCounter + 1;
    tonTimer(IN:=FALSE);
END_IF;

// Use this timer to time out any tests that stall
tonTimer(
    IN:=nTestCounter >= 1,
    PT:=T#2s,
);

METHOD TestParameterCopy
VAR_INPUT
    nTestIndex: UINT;
END_VAR
VAR_INST
    bLocalInit: BOOL := TRUE;
    bAllModified: BOOL;
    bReady: BOOL;
    bDone: BOOL;
END_VAR
TEST(CONCAT('TestParameterCopy', UINT_TO_STRING(nTestIndex)));
IF nTestCounter <> nTestIndex OR bOneTestDone THEN
    RETURN;
END_IF

fbMotionStage(stMotionStage:=stMotionStage);

IF bLocalInit THEN
    stMotionStage.stAxisParametersExposed.bCtrlEnablePosDiffControl     := 100;
    stMotionStage.stAxisParametersExposed.bEncEnableSoftEndMaxControl   := 101;
    stMotionStage.stAxisParametersExposed.bEncEnableSoftEndMinControl   := 102;
    stMotionStage.stAxisParametersExposed.fAccelerationMax              := 103;
    stMotionStage.stAxisParametersExposed.fCtrlPosDiffMax               := 104;
    stMotionStage.stAxisParametersExposed.fCtrlPosDiffMaxTime           := 105;
    stMotionStage.stAxisParametersExposed.fDecelerationMax              := 106;
    stMotionStage.stAxisParametersExposed.fEncSoftEndMax                := 107;
    stMotionStage.stAxisParametersExposed.fEncSoftEndMin                := 108;
    stMotionStage.stAxisParametersExposed.fVeloMaximum                  := 109;
    stMotionStage.stAxisParametersExposed.fEncOffset					:= 110;
    stMotionStage.stAxisParametersExposed.fEncScaleFactorInternal		:= 111;

    bLocalInit := FALSE;

    bAllModified :=
        stMotionStage.stAxisParametersExposed.bCtrlEnablePosDiffControl     <> stMotionStage.stAxisParameters.bCtrlEnablePosDiffControl AND
        stMotionStage.stAxisParametersExposed.bEncEnableSoftEndMaxControl   <> stMotionStage.stAxisParameters.bEncEnableSoftEndMaxControl AND
        stMotionStage.stAxisParametersExposed.bEncEnableSoftEndMinControl   <> stMotionStage.stAxisParameters.bEncEnableSoftEndMinControl AND
        stMotionStage.stAxisParametersExposed.fAccelerationMax              <> stMotionStage.stAxisParameters.fAccelerationMax AND
        stMotionStage.stAxisParametersExposed.fCtrlPosDiffMax               <> stMotionStage.stAxisParameters.fCtrlPosDiffMax AND
        stMotionStage.stAxisParametersExposed.fCtrlPosDiffMaxTime           <> stMotionStage.stAxisParameters.fCtrlPosDiffMaxTime AND
        stMotionStage.stAxisParametersExposed.fDecelerationMax              <> stMotionStage.stAxisParameters.fDecelerationMax AND
        stMotionStage.stAxisParametersExposed.fEncSoftEndMax                <> stMotionStage.stAxisParameters.fEncSoftEndMax AND
        stMotionStage.stAxisParametersExposed.fEncSoftEndMin                <> stMotionStage.stAxisParameters.fEncSoftEndMin AND
        stMotionStage.stAxisParametersExposed.fVeloMaximum                  <> stMotionStage.stAxisParameters.fVeloMaximum AND
        stMotionStage.stAxisParametersExposed.fEncOffset                	<> stMotionStage.stAxisParameters.fEncOffset AND
        stMotionStage.stAxisParametersExposed.fEncScaleFactorInternal       <> stMotionStage.stAxisParameters.fEncScaleFactorInternal;

    AssertTrue(
        Condition:=bAllModified,
        Message:='One or more parameters was not modified initially so the check is invalid.',
    );
END_IF

bReady :=
        stMotionStage.stAxisParameters.bCtrlEnablePosDiffControl     <> 0 AND
        stMotionStage.stAxisParameters.bEncEnableSoftEndMaxControl   <> 0 AND
        stMotionStage.stAxisParameters.bEncEnableSoftEndMinControl   <> 0 AND
        stMotionStage.stAxisParameters.fAccelerationMax              <> 0 AND
        stMotionStage.stAxisParameters.fCtrlPosDiffMax               <> 0 AND
        stMotionStage.stAxisParameters.fCtrlPosDiffMaxTime           <> 0 AND
        stMotionStage.stAxisParameters.fDecelerationMax              <> 0 AND
        stMotionStage.stAxisParameters.fEncSoftEndMax                <> 0 AND
        stMotionStage.stAxisParameters.fEncSoftEndMin                <> 0 AND
        stMotionStage.stAxisParameters.fVeloMaximum                  <> 0 AND
        stMotionStage.stAxisParameters.fEncOffset					 <> 0 AND
        stMotionStage.stAxisParameters.fEncScaleFactorInternal       <> 0;

IF bReady THEN
    bDone :=
        stMotionStage.stAxisParametersExposed.bCtrlEnablePosDiffControl     = stMotionStage.stAxisParameters.bCtrlEnablePosDiffControl AND
        stMotionStage.stAxisParametersExposed.bEncEnableSoftEndMaxControl   = stMotionStage.stAxisParameters.bEncEnableSoftEndMaxControl AND
        stMotionStage.stAxisParametersExposed.bEncEnableSoftEndMinControl   = stMotionStage.stAxisParameters.bEncEnableSoftEndMinControl AND
        stMotionStage.stAxisParametersExposed.fAccelerationMax              = stMotionStage.stAxisParameters.fAccelerationMax AND
        stMotionStage.stAxisParametersExposed.fCtrlPosDiffMax               = stMotionStage.stAxisParameters.fCtrlPosDiffMax AND
        stMotionStage.stAxisParametersExposed.fCtrlPosDiffMaxTime           = stMotionStage.stAxisParameters.fCtrlPosDiffMaxTime AND
        stMotionStage.stAxisParametersExposed.fDecelerationMax              = stMotionStage.stAxisParameters.fDecelerationMax AND
        stMotionStage.stAxisParametersExposed.fEncSoftEndMax                = stMotionStage.stAxisParameters.fEncSoftEndMax AND
        stMotionStage.stAxisParametersExposed.fEncSoftEndMin                = stMotionStage.stAxisParameters.fEncSoftEndMin AND
        stMotionStage.stAxisParametersExposed.fVeloMaximum                  = stMotionStage.stAxisParameters.fVeloMaximum AND
        stMotionStage.stAxisParametersExposed.fEncOffset                	= stMotionStage.stAxisParameters.fEncOffset AND
        stMotionStage.stAxisParametersExposed.fEncScaleFactorInternal       = stMotionStage.stAxisParameters.fEncScaleFactorInternal;
END_IF

IF bDone OR tonTimer.Q THEN
    AssertFalse(
        Condition:=tonTimer.Q,
        Message:=CONCAT(CONCAT('Failed to update the parameters within ', TIME_TO_STRING(tonTimer.PT)),' seconds.'),
    );
    AssertTrue(
        Condition:=bDone,
        Message:='One or more parameters was not copied properly.',
    );

    bOneTestDone := TRUE;
    TEST_FINISHED();
END_IF
END_METHOD

END_FUNCTION_BLOCK

// ---- Tests/Helpers/FB_MotorTestSuite.TcPOU
FUNCTION_BLOCK FB_MotorTestSuite EXTENDS TcUnit.FB_TestSuite
(*
    Base class for motion tests.

    Contains some helper methods that would otherwise need to be instantiated many times,
    but in this form can be accessed quickly and succinctly in the test suite.
*)

METHOD SetEnables
(*
    Set a motion stage's enables such that it is fully allowed to move.
*)
VAR_IN_OUT
    stMotionStage: ST_MotionStage;
END_VAR
stMotionStage.bHardwareEnable := TRUE;
stMotionStage.bLimitBackwardEnable := TRUE;
stMotionStage.bLimitForwardEnable := TRUE;
stMotionStage.bPowerSelf := TRUE;
END_METHOD

METHOD SetEnablesPMPS
(*
    Set a motion stage's enables such that only PMPS would be preventing a move.
*)
VAR_IN_OUT
    stMotionStage: ST_MotionStage;
END_VAR

SetEnables(stMotionStage);
stMotionStage.bPowerSelf := FALSE;
END_METHOD

METHOD SetGoodState
(*
    Mark a state as valid and ready to use.
*)
VAR_IN_OUT
    stPositionState: ST_PositionState;
END_VAR
stPositionState.bMoveOk := TRUE;
stPositionState.bValid := TRUE;
END_METHOD

END_FUNCTION_BLOCK

// ---- Tests/FB_MiscStatesErrorFFO_Test.TcPOU
FUNCTION_BLOCK FB_MiscStatesErrorFFO_Test EXTENDS TcUnit.FB_TestSuite
(*
    Unit tests for FB_MiscStatesErrorFFO
*)
VAR
END_VAR


TestBeamParamsNotOk();
TestZeroRate();
TestUnknownState();
TestTransitionState();
TestDebounce();

METHOD TestBeamParamsNotOk
VAR_INST
    fbMiscFFO: FB_MiscStatesErrorFFO;
    fbArbiter: FB_Arbiter(1);
    fbFFHWO: FB_HardwareFFOutput := (bAutoReset := TRUE);

    stBeamReq: ST_BeamParams;
END_VAR

TEST('TestBeamParamsNotOk');

fbFFHWO.EvaluateOutput();
AssertTrue(
    fbFFHWO.q_xFastFaultOut,
    'Started with a fault',
);

